LIN {X 0,Y 208.214,Z 248.661,A -85,B 0,C 180,E1 -22270.207,E2 -22270.207} C_VEL
LIN {X 0,Y 212.048,Z 236.781,A -85,B 0,C 180,E1 -22272.157,E2 -22272.157} C_VEL
LIN {X 0,Y 215.168,Z 224.656,A -85,B 0,C 180,E1 -22273.649,E2 -22273.649} C_VEL
LIN {X 0,Y 217.166,Z 214.19,A -85,B 0,C 180,E1 -22274.651,E2 -22274.651} C_VEL
LIN {X 0,Y 219.17,Z 200.943,A -85,B 0,C 180,E1 -22275.517,E2 -22275.517} C_VEL
LIN {X 0,Y 220.253,Z 187.914,A -85,B 0,C 180,E1 -22276.059,E2 -22276.059} C_VEL
LIN {X 0,Y 222.25,Z 151.476,A -85,B 0,C 180,E1 -22277.164,E2 -22277.164} C_VEL
LIN {X 0,Y 218.066,Z 142.469,A -85,B 0,C 180,E1 -22278.632,E2 -22278.632} C_VEL
LIN {X 0,Y 210.502,Z 129.434,A -85,B 0,C 180,E1 -22281.386,E2 -22281.386} C_VEL
LIN {X 0,Y 203.081,Z 118.196,A -85,B 0,C 180,E1 -22284.371,E2 -22284.371} C_VEL
LIN {X 0,Y 199.112,Z 112.832,A -85,B 0,C 180,E1 -22286.11,E2 -22286.11} C_VEL
LIN {X 0,Y 196.735,Z 109.497,A -85,B 0,C 180,E1 -22287.228,E2 -22287.228} C_VEL
LIN {X 0,Y 194.076,Z 106.045,A -85,B 0,C 180,E1 -22288.534,E2 -22288.534} C_VEL
LIN {X 0,Y 193.174,Z 104.766,A -85,B 0,C 180,E1 -22289.002,E2 -22289.002} C_VEL
LIN {X 0,Y 190.755,Z 102.14,A -85,B 0,C 180,E1 -22290.255,E2 -22290.255} C_VEL
LIN {X 0,Y 189.444,Z 99.842,A -85,B 0,C 180,E1 -22291.026,E2 -22291.026} C_VEL
LIN {X 0,Y 186.814,Z 97.643,A -85,B 0,C 180,E1 -22292.482,E2 -22292.482} C_VEL
LIN {X 0,Y 185.717,Z 95.405,A -85,B 0,C 180,E1 -22293.22,E2 -22293.22} C_VEL
LIN {X 0,Y 185.515,Z 94.365,A -85,B 0,C 180,E1 -22293.416,E2 -22293.416} C_VEL
LIN {X 0,Y 185.575,Z 94.354,A -85,B 0,C 180,E1 -22297.745,E2 -22297.745} C_VEL
LIN {X 0,Y 185.687,Z 94.337,A -85,B 0,C 180,E1 -22302.374,E2 -22302.374} C_VEL
LIN {X 0,Y 185.724,Z 94.335,A -85,B 0,C 180,E1 -22306.876,E2 -22306.876} C_VEL
LIN {X 0,Y 185.977,Z 94.319,A -85,B 0,C 180,E1 -22311.305,E2 -22311.305} C_VEL
LIN {X 0,Y 186.182,Z 94.286,A -85,B 0,C 180,E1 -22317.836,E2 -22317.836} C_VEL
LIN {X 0,Y 186.383,Z 94.246,A -85,B 0,C 180,E1 -22320,E2 -22320} C_VEL
LIN {X 0,Y 185.889,Z 94.317,A -85,B 0,C 180,E1 -22324.336,E2 -22324.336} C_VEL
LIN {X 0,Y 185.979,Z 94.318,A -85,B 0,C 180,E1 -22328.694,E2 -22328.694} C_VEL
LIN {X 0,Y 185.724,Z 94.335,A -85,B 0,C 180,E1 -22333.123,E2 -22333.123} C_VEL
LIN {X 0,Y 185.687,Z 94.336,A -85,B 0,C 180,E1 -22337.625,E2 -22337.625} C_VEL
LIN {X 0,Y 185.598,Z 94.35,A -85,B 0,C 180,E1 -22342.251,E2 -22342.251} C_VEL
LIN {X 0,Y 185.565,Z 94.357,A -85,B 0,C 180,E1 -22347.031,E2 -22347.031} C_VEL
LIN {X 0,Y 185.584,Z 94.473,A -85,B 0,C 180,E1 -22350.274,E2 -22350.274} C_VEL
LIN {X 0,Y 186.862,Z 98.544,A -85,B 0,C 180,E1 -22354.033,E2 -22354.033} C_VEL
LIN {X 0,Y 189.971,Z 103.26,A -85,B 0,C 180,E1 -22355.883,E2 -22355.883} C_VEL
LIN {X 0,Y 191.772,Z 105.585,A -85,B 0,C 180,E1 -22356.86,E2 -22356.86} C_VEL
LIN {X 0,Y 195.084,Z 110.421,A -85,B 0,C 180,E1 -22358.586,E2 -22358.586} C_VEL
LIN {X 0,Y 200.019,Z 118.409,A -85,B 0,C 180,E1 -22360.974,E2 -22360.974} C_VEL
LIN {X 0,Y 203.707,Z 124.608,A -85,B 0,C 180,E1 -22362.617,E2 -22362.617} C_VEL
LIN {X 0,Y 209.57,Z 135.23,A -85,B 0,C 180,E1 -22365.047,E2 -22365.047} C_VEL
LIN {X 0,Y 215.403,Z 147.492,A -85,B 0,C 180,E1 -22367.312,E2 -22367.312} C_VEL
LIN {X 0,Y 220.114,Z 159.014,A -85,B 0,C 180,E1 -22369.064,E2 -22369.064} C_VEL
LIN {X 0,Y 221.3,Z 169.331,A -85,B 0,C 180,E1 -22369.809,E2 -22369.809} C_VEL
LIN {X 0,Y 220.488,Z 184.555,A -85,B 0,C 180,E1 -22370.276,E2 -22370.276} C_VEL
LIN {X 0,Y 219.649,Z 190.415,A -85,B 0,C 180,E1 -22370.315,E2 -22370.315} C_VEL
LIN {X 0,Y 214.146,Z 209.415,A -85,B 0,C 180,E1 -22369.874,E2 -22369.874} C_VEL
LIN {X 0,Y 213.002,Z 215.173,A -85,B 0,C 180,E1 -22370.032,E2 -22370.032} C_VEL
LIN {X 0,Y 210.897,Z 228.271,A -85,B 0,C 180,E1 -22370.869,E2 -22370.869} C_VEL
LIN {X 0,Y 208.139,Z 240.343,A -85,B 0,C 180,E1 -22371.958,E2 -22371.958} C_VEL
LIN {X 0,Y 204.723,Z 251.98,A -85,B 0,C 180,E1 -22373.382,E2 -22373.382} C_VEL
LIN {X 0,Y 201.939,Z 260.097,A -85,B 0,C 180,E1 -22374.648,E2 -22374.648} C_VEL
LIN {X 0,Y 198.09,Z 270.178,A -85,B 0,C 180,E1 -22376.638,E2 -22376.638} C_VEL
LIN {X 0,Y 194.028,Z 279.294,A -85,B 0,C 180,E1 -22378.924,E2 -22378.924} C_VEL
LIN {X 0,Y 189.721,Z 288.196,A -85,B 0,C 180,E1 -22381.815,E2 -22381.815} C_VEL
LIN {X 0,Y 186.057,Z 295.38,A -85,B 0,C 180,E1 -22384.852,E2 -22384.852} C_VEL
LIN {X 0,Y 182.517,Z 301.95,A -85,B 0,C 180,E1 -22388.542,E2 -22388.542} C_VEL
LIN {X 0,Y 180.008,Z 306.321,A -85,B 0,C 180,E1 -22391.799,E2 -22391.799} C_VEL
LIN {X 0,Y 178.619,Z 308.644,A -85,B 0,C 180,E1 -22394.012,E2 -22394.012} C_VEL
LIN {X 0,Y 177.62,Z 310.548,A -85,B 0,C 180,E1 -22396.266,E2 -22396.266} C_VEL
LIN {X 0,Y 176.909,Z 311.998,A -85,B 0,C 180,E1 -22398.542,E2 -22398.542} C_VEL
LIN {X 0,Y 176.122,Z 313.708,A -85,B 0,C 180,E1 -22403.124,E2 -22403.124} C_VEL
LIN {X 0,Y 176.059,Z 313.961,A -85,B 0,C 180,E1 -22406.336,E2 -22406.336} C_VEL
LIN {X 0,Y 176.324,Z 313.298,A -85,B 0,C 180,E1 -22409.999,E2 -22409.999} C_VEL
LIN {X 0,Y 176.146,Z 311.28,A -85,B 0,C 180,E1 -22414.08,E2 -22414.08} C_VEL
LIN {X 0,Y 176.25,Z 308.042,A -85,B 0,C 180,E1 -22418.022,E2 -22418.022} C_VEL
LIN {X 0,Y 176.795,Z 304.072,A -85,B 0,C 180,E1 -22421.464,E2 -22421.464} C_VEL
LIN {X 0,Y 178.094,Z 297.957,A -85,B 0,C 180,E1 -22425.448,E2 -22425.448} C_VEL
LIN {X 0,Y 179.851,Z 291.253,A -85,B 0,C 180,E1 -22428.806,E2 -22428.806} C_VEL
LIN {X 0,Y 181.508,Z 285.685,A -85,B 0,C 180,E1 -22431.088,E2 -22431.088} C_VEL
LIN {X 0,Y 183.867,Z 276.18,A -85,B 0,C 180,E1 -22434.261,E2 -22434.261} C_VEL
LIN {X 0,Y 186.685,Z 266.151,A -85,B 0,C 180,E1 -22436.856,E2 -22436.856} C_VEL
LIN {X 0,Y 189.57,Z 254.816,A -85,B 0,C 180,E1 -22439.116,E2 -22439.116} C_VEL
LIN {X 0,Y 191.94,Z 243.68,A -85,B 0,C 180,E1 -22440.838,E2 -22440.838} C_VEL
LIN {X 0,Y 194.237,Z 231.337,A -85,B 0,C 180,E1 -22442.255,E2 -22442.255} C_VEL
LIN {X 0,Y 195.884,Z 218.597,A -85,B 0,C 180,E1 -22443.292,E2 -22443.292} C_VEL
LIN {X 0,Y 196.941,Z 205.474,A -85,B 0,C 180,E1 -22443.971,E2 -22443.971} C_VEL
LIN {X 0,Y 198.808,Z 161.492,A -85,B 0,C 180,E1 -22445.49,E2 -22445.49} C_VEL
LIN {X 0,Y 196.398,Z 137.184,A -85,B 0,C 180,E1 -22446.97,E2 -22446.97} C_VEL
LIN {X 0,Y 189.853,Z 120.576,A -85,B 0,C 180,E1 -22449.039,E2 -22449.039} C_VEL
LIN {X 0,Y 184.006,Z 108.494,A -85,B 0,C 180,E1 -22450.928,E2 -22450.928} C_VEL
LIN {X 0,Y 181.537,Z 103.873,A -85,B 0,C 180,E1 -22451.754,E2 -22451.754} C_VEL
LIN {X 0,Y 179.702,Z 100.17,A -85,B 0,C 180,E1 -22452.423,E2 -22452.423} C_VEL
LIN {X 0,Y 178.389,Z 95.265,A -85,B 0,C 180,E1 -22455.595,E2 -22455.595} C_VEL
LIN {X 0,Y 178.401,Z 95.258,A -85,B 0,C 180,E1 -22458.459,E2 -22458.459} C_VEL
LIN {X 0,Y 178.421,Z 95.248,A -85,B 0,C 180,E1 -22463.783,E2 -22463.783} C_VEL
LIN {X 0,Y 178.486,Z 95.25,A -85,B 0,C 180,E1 -22466.547,E2 -22466.547} C_VEL
LIN {X 0,Y 178.522,Z 95.247,A -85,B 0,C 180,E1 -22470.006,E2 -22470.006} C_VEL
LIN {X 0,Y 178.533,Z 95.24,A -85,B 0,C 180,E1 -22474.876,E2 -22474.876} C_VEL
LIN {X 0,Y 178.622,Z 95.22,A -85,B 0,C 180,E1 -22480.784,E2 -22480.784} C_VEL
LIN {X 0,Y 178.659,Z 95.214,A -85,B 0,C 180,E1 -22486.348,E2 -22486.348} C_VEL
LIN {X 0,Y 178.911,Z 95.199,A -85,B 0,C 180,E1 -22490.96,E2 -22490.96} C_VEL
LIN {X 0,Y 179.15,Z 95.157,A -85,B 0,C 180,E1 -22497.752,E2 -22497.752} C_VEL
LIN {X 0,Y 179.367,Z 95.142,A -85,B 0,C 180,E1 -22500,E2 -22500} C_VEL
LIN {X 0,Y 178.857,Z 95.184,A -85,B 0,C 180,E1 -22504.508,E2 -22504.508} C_VEL
LIN {X 0,Y 178.908,Z 95.196,A -85,B 0,C 180,E1 -22509.041,E2 -22509.041} C_VEL
LIN {X 0,Y 178.655,Z 95.209,A -85,B 0,C 180,E1 -22513.653,E2 -22513.653} C_VEL
LIN {X 0,Y 178.623,Z 95.225,A -85,B 0,C 180,E1 -22519.217,E2 -22519.217} C_VEL
LIN {X 0,Y 178.534,Z 95.245,A -85,B 0,C 180,E1 -22525.125,E2 -22525.125} C_VEL
LIN {X 0,Y 178.477,Z 95.25,A -85,B 0,C 180,E1 -22530.792,E2 -22530.792} C_VEL
LIN {X 0,Y 178.484,Z 95.251,A -85,B 0,C 180,E1 -22534.22,E2 -22534.22} C_VEL
LIN {X 0,Y 178.388,Z 95.265,A -85,B 0,C 180,E1 -22539.077,E2 -22539.077} C_VEL
LIN {X 0,Y 178.394,Z 95.262,A -85,B 0,C 180,E1 -22542.047,E2 -22542.047} C_VEL
LIN {X 0,Y 178.393,Z 95.263,A -85,B 0,C 180,E1 -22545.165,E2 -22545.165} C_VEL
LIN {X 0,Y 178.4,Z 95.263,A -85,B 0,C 180,E1 -22548.462,E2 -22548.462} C_VEL
LIN {X 0,Y 178.42,Z 95.261,A -85,B 0,C 180,E1 -22553.783,E2 -22553.783} C_VEL
LIN {X 0,Y 178.464,Z 95.409,A -85,B 0,C 180,E1 -22554.734,E2 -22554.734} C_VEL
LIN {X 0,Y 179.354,Z 97.939,A -85,B 0,C 180,E1 -22555.095,E2 -22555.095} C_VEL
LIN {X 0,Y 181.323,Z 100.58,A -85,B 0,C 180,E1 -22555.729,E2 -22555.729} C_VEL
LIN {X 0,Y 188.55,Z 112.687,A -85,B 0,C 180,E1 -22558.014,E2 -22558.014} C_VEL
LIN {X 0,Y 194.723,Z 124.313,A -85,B 0,C 180,E1 -22559.841,E2 -22559.841} C_VEL
LIN {X 0,Y 200.072,Z 136.131,A -85,B 0,C 180,E1 -22561.378,E2 -22561.378} C_VEL
LIN {X 0,Y 197.219,Z 194.928,A -85,B 0,C 180,E1 -22563.391,E2 -22563.391} C_VEL
LIN {X 0,Y 196.004,Z 208.238,A -85,B 0,C 180,E1 -22564.245,E2 -22564.245} C_VEL
LIN {X 0,Y 194.445,Z 220.579,A -85,B 0,C 180,E1 -22565.44,E2 -22565.44} C_VEL
LIN {X 0,Y 192.613,Z 231.72,A -85,B 0,C 180,E1 -22566.907,E2 -22566.907} C_VEL
LIN {X 0,Y 190.187,Z 243.267,A -85,B 0,C 180,E1 -22568.883,E2 -22568.883} C_VEL
LIN {X 0,Y 187.654,Z 253.66,A -85,B 0,C 180,E1 -22571.155,E2 -22571.155} C_VEL
LIN {X 0,Y 185.261,Z 262.174,A -85,B 0,C 180,E1 -22573.471,E2 -22573.471} C_VEL
LIN {X 0,Y 183.031,Z 270.012,A -85,B 0,C 180,E1 -22576.115,E2 -22576.115} C_VEL
LIN {X 0,Y 180.759,Z 277.681,A -85,B 0,C 180,E1 -22579.358,E2 -22579.358} C_VEL
LIN {X 0,Y 178.796,Z 284.725,A -85,B 0,C 180,E1 -22583.228,E2 -22583.228} C_VEL
LIN {X 0,Y 177.53,Z 289.43,A -85,B 0,C 180,E1 -22586.596,E2 -22586.596} C_VEL
LIN {X 0,Y 176.737,Z 293.036,A -85,B 0,C 180,E1 -22590.001,E2 -22590.001} C_VEL
LIN {X 0,Y 176.474,Z 294.901,A -85,B 0,C 180,E1 -22592.283,E2 -22592.283} C_VEL
LIN {X 0,Y 176.362,Z 296.496,A -85,B 0,C 180,E1 -22594.957,E2 -22594.957} C_VEL
LIN {X 0,Y 176.247,Z 297.954,A -85,B 0,C 180,E1 -22599.179,E2 -22599.179} C_VEL
LIN {X 0,Y 176.415,Z 298.2,A -85,B 0,C 180,E1 -22601.49,E2 -22601.49} C_VEL
LIN {X 0,Y 177.52,Z 297.423,A -85,B 0,C 180,E1 -22606.09,E2 -22606.09} C_VEL
LIN {X 0,Y 178.83,Z 295.862,A -85,B 0,C 180,E1 -22609.402,E2 -22609.402} C_VEL
LIN {X 0,Y 181.422,Z 292.147,A -85,B 0,C 180,E1 -22614.002,E2 -22614.002} C_VEL
LIN {X 0,Y 183.963,Z 288.165,A -85,B 0,C 180,E1 -22617.287,E2 -22617.287} C_VEL
LIN {X 0,Y 187.506,Z 282.086,A -85,B 0,C 180,E1 -22620.96,E2 -22620.96} C_VEL
LIN {X 0,Y 191.247,Z 275.216,A -85,B 0,C 180,E1 -22624.085,E2 -22624.085} C_VEL
LIN {X 0,Y 195.437,Z 266.754,A -85,B 0,C 180,E1 -22627.038,E2 -22627.038} C_VEL
LIN {X 0,Y 199.065,Z 257.983,A -85,B 0,C 180,E1 -22629.457,E2 -22629.457} C_VEL
LIN {X 0,Y 203.193,Z 247.149,A -85,B 0,C 180,E1 -22631.746,E2 -22631.746} C_VEL
LIN {X 0,Y 206.781,Z 236.268,A -85,B 0,C 180,E1 -22633.493,E2 -22633.493} C_VEL
LIN {X 0,Y 209.932,Z 224.261,A -85,B 0,C 180,E1 -22634.963,E2 -22634.963} C_VEL
LIN {X 0,Y 211.803,Z 214.817,A -85,B 0,C 180,E1 -22635.876,E2 -22635.876} C_VEL
LIN {X 0,Y 213.894,Z 201.6,A -85,B 0,C 180,E1 -22636.756,E2 -22636.756} C_VEL
LIN {X 0,Y 215.06,Z 188.275,A -85,B 0,C 180,E1 -22637.324,E2 -22637.324} C_VEL
LIN {X 0,Y 217.077,Z 153.919,A -85,B 0,C 180,E1 -22638.368,E2 -22638.368} C_VEL
LIN {X 0,Y 213.436,Z 146.148,A -85,B 0,C 180,E1 -22639.719,E2 -22639.719} C_VEL
LIN {X 0,Y 206.422,Z 134.012,A -85,B 0,C 180,E1 -22642.416,E2 -22642.416} C_VEL
LIN {X 0,Y 199.687,Z 123.62,A -85,B 0,C 180,E1 -22645.274,E2 -22645.274} C_VEL
LIN {X 0,Y 195.646,Z 117.975,A -85,B 0,C 180,E1 -22647.147,E2 -22647.147} C_VEL
LIN {X 0,Y 193.419,Z 114.948,A -85,B 0,C 180,E1 -22648.247,E2 -22648.247} C_VEL
LIN {X 0,Y 190.362,Z 110.778,A -85,B 0,C 180,E1 -22649.853,E2 -22649.853} C_VEL
LIN {X 0,Y 187.716,Z 107.553,A -85,B 0,C 180,E1 -22651.318,E2 -22651.318} C_VEL
LIN {X 0,Y 186.732,Z 106.033,A -85,B 0,C 180,E1 -22651.912,E2 -22651.912} C_VEL
LIN {X 0,Y 184.168,Z 103.462,A -85,B 0,C 180,E1 -22653.435,E2 -22653.435} C_VEL
LIN {X 0,Y 182.822,Z 100.932,A -85,B 0,C 180,E1 -22654.375,E2 -22654.375} C_VEL
LIN {X 0,Y 180.167,Z 98.955,A -85,B 0,C 180,E1 -22656.103,E2 -22656.103} C_VEL
LIN {X 0,Y 178.891,Z 96.811,A -85,B 0,C 180,E1 -22657.096,E2 -22657.096} C_VEL
LIN {X 0,Y 178.539,Z 95.229,A -85,B 0,C 180,E1 -22657.583,E2 -22657.583} C_VEL
LIN {X 0,Y 178.641,Z 95.216,A -85,B 0,C 180,E1 -22661.655,E2 -22661.655} C_VEL
LIN {X 0,Y 178.652,Z 95.22,A -85,B 0,C 180,E1 -22666.347,E2 -22666.347} C_VEL
LIN {X 0,Y 178.908,Z 95.2,A -85,B 0,C 180,E1 -22670.959,E2 -22670.959} C_VEL
LIN {X 0,Y 179.13,Z 95.165,A -85,B 0,C 180,E1 -22677.751,E2 -22677.751} C_VEL
LIN {X 0,Y 179.348,Z 95.122,A -85,B 0,C 180,E1 -22680,E2 -22680} C_VEL
LIN {X 0,Y 178.838,Z 95.193,A -85,B 0,C 180,E1 -22684.507,E2 -22684.507} C_VEL
LIN {X 0,Y 178.909,Z 95.199,A -85,B 0,C 180,E1 -22689.04,E2 -22689.04} C_VEL
LIN {X 0,Y 178.652,Z 95.221,A -85,B 0,C 180,E1 -22693.652,E2 -22693.652} C_VEL
LIN {X 0,Y 178.625,Z 95.229,A -85,B 0,C 180,E1 -22699.215,E2 -22699.215} C_VEL
LIN {X 0,Y 178.537,Z 95.243,A -85,B 0,C 180,E1 -22705.124,E2 -22705.124} C_VEL
LIN {X 0,Y 178.515,Z 95.236,A -85,B 0,C 180,E1 -22706.92,E2 -22706.92} C_VEL
LIN {X 0,Y 179.396,Z 97.872,A -85,B 0,C 180,E1 -22709.746,E2 -22709.746} C_VEL
LIN {X 0,Y 182.55,Z 102.601,A -85,B 0,C 180,E1 -22712.028,E2 -22712.028} C_VEL
LIN {X 0,Y 184.519,Z 105.013,A -85,B 0,C 180,E1 -22713.295,E2 -22713.295} C_VEL
LIN {X 0,Y 188.306,Z 110.4,A -85,B 0,C 180,E1 -22715.59,E2 -22715.59} C_VEL
LIN {X 0,Y 192.963,Z 117.683,A -85,B 0,C 180,E1 -22718.16,E2 -22718.16} C_VEL
LIN {X 0,Y 197.039,Z 124.388,A -85,B 0,C 180,E1 -22720.206,E2 -22720.206} C_VEL
LIN {X 0,Y 201.68,Z 132.442,A -85,B 0,C 180,E1 -22722.352,E2 -22722.352} C_VEL
LIN {X 0,Y 207.554,Z 143.812,A -85,B 0,C 180,E1 -22724.866,E2 -22724.866} C_VEL
LIN {X 0,Y 213.318,Z 157.114,A -85,B 0,C 180,E1 -22727.195,E2 -22727.195} C_VEL
LIN {X 0,Y 215.175,Z 161.886,A -85,B 0,C 180,E1 -22727.921,E2 -22727.921} C_VEL
LIN {X 0,Y 216.084,Z 170.94,A -85,B 0,C 180,E1 -22728.576,E2 -22728.576} C_VEL
LIN {X 0,Y 213.683,Z 209.608,A -85,B 0,C 180,E1 -22729.791,E2 -22729.791} C_VEL
LIN {X 0,Y 213.002,Z 215.173,A -85,B 0,C 180,E1 -22730.032,E2 -22730.032} C_VEL
LIN {X 0,Y 212.19,Z 218.992,A -85,B 0,C 180,E1 -22730.167,E2 -22730.167} C_VEL
LIN {X 0,Y 209.468,Z 226.416,A -85,B 0,C 180,E1 -22730.29,E2 -22730.29} C_VEL
LIN {X 0,Y 203.966,Z 238.08,A -85,B 0,C 180,E1 -22730.587,E2 -22730.587} C_VEL
LIN {X 0,Y 201.638,Z 244.264,A -85,B 0,C 180,E1 -22731.113,E2 -22731.113} C_VEL
LIN {X 0,Y 198.06,Z 255.152,A -85,B 0,C 180,E1 -22732.578,E2 -22732.578} C_VEL
LIN {X 0,Y 193.935,Z 266.11,A -85,B 0,C 180,E1 -22734.561,E2 -22734.561} C_VEL
LIN {X 0,Y 189.672,Z 275.927,A -85,B 0,C 180,E1 -22736.869,E2 -22736.869} C_VEL
LIN {X 0,Y 185.67,Z 283.993,A -85,B 0,C 180,E1 -22739.269,E2 -22739.269} C_VEL
LIN {X 0,Y 181.418,Z 291.932,A -85,B 0,C 180,E1 -22742.297,E2 -22742.297} C_VEL
LIN {X 0,Y 178.037,Z 298.141,A -85,B 0,C 180,E1 -22745.403,E2 -22745.403} C_VEL
LIN {X 0,Y 174.926,Z 303.391,A -85,B 0,C 180,E1 -22748.801,E2 -22748.801} C_VEL
LIN {X 0,Y 172.511,Z 307.361,A -85,B 0,C 180,E1 -22752.208,E2 -22752.208} C_VEL
LIN {X 0,Y 170.684,Z 310.316,A -85,B 0,C 180,E1 -22755.696,E2 -22755.696} C_VEL
LIN {X 0,Y 169.355,Z 312.766,A -85,B 0,C 180,E1 -22760.444,E2 -22760.444} C_VEL
LIN {X 0,Y 168.966,Z 313.672,A -85,B 0,C 180,E1 -22765.227,E2 -22765.227} C_VEL
LIN {X 0,Y 169.054,Z 313.501,A -85,B 0,C 180,E1 -22767.617,E2 -22767.617} C_VEL
LIN {X 0,Y 169.24,Z 312.933,A -85,B 0,C 180,E1 -22769.999,E2 -22769.999} C_VEL
LIN {X 0,Y 169.056,Z 311.115,A -85,B 0,C 180,E1 -22773.863,E2 -22773.863} C_VEL
LIN {X 0,Y 169.185,Z 307.6,A -85,B 0,C 180,E1 -22778.359,E2 -22778.359} C_VEL
LIN {X 0,Y 169.78,Z 303.588,A -85,B 0,C 180,E1 -22781.944,E2 -22781.944} C_VEL
LIN {X 0,Y 171.235,Z 297.41,A -85,B 0,C 180,E1 -22786.083,E2 -22786.083} C_VEL
LIN {X 0,Y 173.109,Z 290.654,A -85,B 0,C 180,E1 -22789.568,E2 -22789.568} C_VEL
LIN {X 0,Y 174.701,Z 285.446,A -85,B 0,C 180,E1 -22791.777,E2 -22791.777} C_VEL
LIN {X 0,Y 176.871,Z 277.26,A -85,B 0,C 180,E1 -22794.658,E2 -22794.658} C_VEL
LIN {X 0,Y 179.713,Z 267.506,A -85,B 0,C 180,E1 -22797.355,E2 -22797.355} C_VEL
LIN {X 0,Y 182.663,Z 256.674,A -85,B 0,C 180,E1 -22799.693,E2 -22799.693} C_VEL
LIN {X 0,Y 185.094,Z 246.118,A -85,B 0,C 180,E1 -22801.472,E2 -22801.472} C_VEL
LIN {X 0,Y 187.645,Z 233.414,A -85,B 0,C 180,E1 -22803.053,E2 -22803.053} C_VEL
LIN {X 0,Y 189.537,Z 220.471,A -85,B 0,C 180,E1 -22804.216,E2 -22804.216} C_VEL
LIN {X 0,Y 190.723,Z 207.67,A -85,B 0,C 180,E1 -22804.961,E2 -22804.961} C_VEL
LIN {X 0,Y 192.809,Z 162.477,A -85,B 0,C 180,E1 -22806.567,E2 -22806.567} C_VEL
LIN {X 0,Y 190.647,Z 139.752,A -85,B 0,C 180,E1 -22808.004,E2 -22808.004} C_VEL
LIN {X 0,Y 185.116,Z 125.198,A -85,B 0,C 180,E1 -22809.873,E2 -22809.873} C_VEL
LIN {X 0,Y 179.303,Z 112.892,A -85,B 0,C 180,E1 -22811.865,E2 -22811.865} C_VEL
LIN {X 0,Y 174.268,Z 103.614,A -85,B 0,C 180,E1 -22813.673,E2 -22813.673} C_VEL
LIN {X 0,Y 172.282,Z 99.694,A -85,B 0,C 180,E1 -22814.494,E2 -22814.494} C_VEL
LIN {X 0,Y 171.354,Z 96.14,A -85,B 0,C 180,E1 -22816.917,E2 -22816.917} C_VEL
LIN {X 0,Y 171.363,Z 96.108,A -85,B 0,C 180,E1 -22822.035,E2 -22822.035} C_VEL
LIN {X 0,Y 171.397,Z 96.134,A -85,B 0,C 180,E1 -22825.092,E2 -22825.092} C_VEL
LIN {X 0,Y 171.448,Z 96.129,A -85,B 0,C 180,E1 -22830.535,E2 -22830.535} C_VEL
LIN {X 0,Y 171.457,Z 96.127,A -85,B 0,C 180,E1 -22835.802,E2 -22835.802} C_VEL
LIN {X 0,Y 171.578,Z 96.097,A -85,B 0,C 180,E1 -22840.872,E2 -22840.872} C_VEL
LIN {X 0,Y 171.577,Z 96.101,A -85,B 0,C 180,E1 -22845.773,E2 -22845.773} C_VEL
LIN {X 0,Y 171.847,Z 96.075,A -85,B 0,C 180,E1 -22850.585,E2 -22850.585} C_VEL
LIN {X 0,Y 171.811,Z 96.066,A -85,B 0,C 180,E1 -22855.308,E2 -22855.308} C_VEL
LIN {X 0,Y 172.33,Z 96.018,A -85,B 0,C 180,E1 -22860.001,E2 -22860.001} C_VEL
LIN {X 0,Y 171.805,Z 96.061,A -85,B 0,C 180,E1 -22864.693,E2 -22864.693} C_VEL
LIN {X 0,Y 171.845,Z 96.077,A -85,B 0,C 180,E1 -22869.416,E2 -22869.416} C_VEL
LIN {X 0,Y 171.573,Z 96.093,A -85,B 0,C 180,E1 -22874.228,E2 -22874.228} C_VEL
LIN {X 0,Y 171.545,Z 96.104,A -85,B 0,C 180,E1 -22879.563,E2 -22879.563} C_VEL
LIN {X 0,Y 171.469,Z 96.125,A -85,B 0,C 180,E1 -22885.617,E2 -22885.617} C_VEL
LIN {X 0,Y 171.44,Z 96.127,A -85,B 0,C 180,E1 -22890.587,E2 -22890.587} C_VEL
LIN {X 0,Y 171.392,Z 96.133,A -85,B 0,C 180,E1 -22895.036,E2 -22895.036} C_VEL
LIN {X 0,Y 171.344,Z 96.14,A -85,B 0,C 180,E1 -22898.803,E2 -22898.803} C_VEL
LIN {X 0,Y 171.319,Z 96.144,A -85,B 0,C 180,E1 -22904.219,E2 -22904.219} C_VEL
LIN {X 0,Y 171.332,Z 96.144,A -85,B 0,C 180,E1 -22908.981,E2 -22908.981} C_VEL
LIN {X 0,Y 171.348,Z 96.148,A -85,B 0,C 180,E1 -22912.791,E2 -22912.791} C_VEL
LIN {X 0,Y 172.434,Z 99.112,A -85,B 0,C 180,E1 -22913.268,E2 -22913.268} C_VEL
LIN {X 0,Y 174.241,Z 101.349,A -85,B 0,C 180,E1 -22913.898,E2 -22913.898} C_VEL
LIN {X 0,Y 176.435,Z 104.7,A -85,B 0,C 180,E1 -22914.673,E2 -22914.673} C_VEL
LIN {X 0,Y 183.024,Z 115.736,A -85,B 0,C 180,E1 -22916.888,E2 -22916.888} C_VEL
LIN {X 0,Y 189.243,Z 127.483,A -85,B 0,C 180,E1 -22918.845,E2 -22918.845} C_VEL
LIN {X 0,Y 194.018,Z 137.872,A -85,B 0,C 180,E1 -22920.294,E2 -22920.294} C_VEL
LIN {X 0,Y 191.167,Z 194.962,A -85,B 0,C 180,E1 -22922.297,E2 -22922.297} C_VEL
LIN {X 0,Y 189.934,Z 208.269,A -85,B 0,C 180,E1 -22923.169,E2 -22923.169} C_VEL
LIN {X 0,Y 188.241,Z 221,A -85,B 0,C 180,E1 -22924.426,E2 -22924.426} C_VEL
LIN {X 0,Y 186.15,Z 232.898,A -85,B 0,C 180,E1 -22926.056,E2 -22926.056} C_VEL
LIN {X 0,Y 183.624,Z 244.288,A -85,B 0,C 180,E1 -22928.089,E2 -22928.089} C_VEL
LIN {X 0,Y 180.983,Z 254.561,A -85,B 0,C 180,E1 -22930.432,E2 -22930.432} C_VEL
LIN {X 0,Y 178.5,Z 262.976,A -85,B 0,C 180,E1 -22932.826,E2 -22932.826} C_VEL
LIN {X 0,Y 175.779,Z 272.078,A -85,B 0,C 180,E1 -22936.121,E2 -22936.121} C_VEL
LIN {X 0,Y 173.468,Z 279.413,A -85,B 0,C 180,E1 -22939.496,E2 -22939.496} C_VEL
LIN {X 0,Y 171.775,Z 285.291,A -85,B 0,C 180,E1 -22942.95,E2 -22942.95} C_VEL
LIN {X 0,Y 170.445,Z 289.945,A -85,B 0,C 180,E1 -22946.455,E2 -22946.455} C_VEL
LIN {X 0,Y 169.656,Z 293.501,A -85,B 0,C 180,E1 -22950.001,E2 -22950.001} C_VEL
LIN {X 0,Y 169.384,Z 295.33,A -85,B 0,C 180,E1 -22952.379,E2 -22952.379} C_VEL
LIN {X 0,Y 169.289,Z 296.76,A -85,B 0,C 180,E1 -22954.884,E2 -22954.884} C_VEL
LIN {X 0,Y 169.188,Z 298.31,A -85,B 0,C 180,E1 -22959.565,E2 -22959.565} C_VEL
LIN {X 0,Y 169.401,Z 298.519,A -85,B 0,C 180,E1 -22961.973,E2 -22961.973} C_VEL
LIN {X 0,Y 170.627,Z 297.691,A -85,B 0,C 180,E1 -22966.758,E2 -22966.758} C_VEL
LIN {X 0,Y 171.922,Z 296.261,A -85,B 0,C 180,E1 -22969.909,E2 -22969.909} C_VEL
LIN {X 0,Y 174.071,Z 293.388,A -85,B 0,C 180,E1 -22973.813,E2 -22973.813} C_VEL
LIN {X 0,Y 176.597,Z 289.721,A -85,B 0,C 180,E1 -22977.237,E2 -22977.237} C_VEL
LIN {X 0,Y 179.678,Z 284.827,A -85,B 0,C 180,E1 -22980.624,E2 -22980.624} C_VEL
LIN {X 0,Y 183.312,Z 278.804,A -85,B 0,C 180,E1 -22983.775,E2 -22983.775} C_VEL
LIN {X 0,Y 187.459,Z 271.177,A -85,B 0,C 180,E1 -22986.86,E2 -22986.86} C_VEL
LIN {X 0,Y 191.611,Z 262.34,A -85,B 0,C 180,E1 -22989.623,E2 -22989.623} C_VEL
LIN {X 0,Y 195.688,Z 252.605,A -85,B 0,C 180,E1 -22991.984,E2 -22991.984} C_VEL
LIN {X 0,Y 199.765,Z 241.619,A -85,B 0,C 180,E1 -22994.015,E2 -22994.015} C_VEL
LIN {X 0,Y 203.067,Z 230.797,A -85,B 0,C 180,E1 -22995.547,E2 -22995.547} C_VEL
LIN {X 0,Y 205.919,Z 218.39,A -85,B 0,C 180,E1 -22996.915,E2 -22996.915} C_VEL
LIN {X 0,Y 208.258,Z 205.643,A -85,B 0,C 180,E1 -22997.871,E2 -22997.871} C_VEL
LIN {X 0,Y 209.754,Z 191.86,A -85,B 0,C 180,E1 -22998.538,E2 -22998.538} C_VEL
LIN {X 0,Y 211.924,Z 156.256,A -85,B 0,C 180,E1 -22999.659,E2 -22999.659} C_VEL
LIN {X 0,Y 208.539,Z 149.298,A -85,B 0,C 180,E1 -23000.983,E2 -23000.983} C_VEL
LIN {X 0,Y 202.366,Z 138.531,A -85,B 0,C 180,E1 -23003.505,E2 -23003.505} C_VEL
LIN {X 0,Y 196.398,Z 129.041,A -85,B 0,C 180,E1 -23006.189,E2 -23006.189} C_VEL
LIN {X 0,Y 190.681,Z 120.93,A -85,B 0,C 180,E1 -23009.038,E2 -23009.038} C_VEL
LIN {X 0,Y 187.427,Z 116.547,A -85,B 0,C 180,E1 -23010.825,E2 -23010.825} C_VEL
LIN {X 0,Y 184.56,Z 112.583,A -85,B 0,C 180,E1 -23012.539,E2 -23012.539} C_VEL
LIN {X 0,Y 181.574,Z 109.281,A -85,B 0,C 180,E1 -23014.417,E2 -23014.417} C_VEL
LIN {X 0,Y 180.462,Z 107.364,A -85,B 0,C 180,E1 -23015.218,E2 -23015.218} C_VEL
LIN {X 0,Y 177.688,Z 104.843,A -85,B 0,C 180,E1 -23017.162,E2 -23017.162} C_VEL
LIN {X 0,Y 176.125,Z 101.923,A -85,B 0,C 180,E1 -23018.492,E2 -23018.492} C_VEL
LIN {X 0,Y 173.471,Z 100.142,A -85,B 0,C 180,E1 -23020.646,E2 -23020.646} C_VEL
LIN {X 0,Y 171.913,Z 97.508,A -85,B 0,C 180,E1 -23022.221,E2 -23022.221} C_VEL
LIN {X 0,Y 171.573,Z 96.095,A -85,B 0,C 180,E1 -23022.723,E2 -23022.723} C_VEL
LIN {X 0,Y 171.771,Z 96.072,A -85,B 0,C 180,E1 -23029.105,E2 -23029.105} C_VEL
LIN {X 0,Y 171.862,Z 96.058,A -85,B 0,C 180,E1 -23032.953,E2 -23032.953} C_VEL
LIN {X 0,Y 172.078,Z 96.044,A -85,B 0,C 180,E1 -23037.659,E2 -23037.659} C_VEL
LIN {X 0,Y 172.313,Z 95.998,A -85,B 0,C 180,E1 -23039.999,E2 -23039.999} C_VEL
LIN {X 0,Y 171.788,Z 96.069,A -85,B 0,C 180,E1 -23044.693,E2 -23044.693} C_VEL
LIN {X 0,Y 171.847,Z 96.075,A -85,B 0,C 180,E1 -23049.415,E2 -23049.415} C_VEL
LIN {X 0,Y 171.57,Z 96.11,A -85,B 0,C 180,E1 -23054.227,E2 -23054.227} C_VEL
LIN {X 0,Y 171.547,Z 96.114,A -85,B 0,C 180,E1 -23059.561,E2 -23059.561} C_VEL
LIN {X 0,Y 171.476,Z 96.224,A -85,B 0,C 180,E1 -23063.074,E2 -23063.074} C_VEL
LIN {X 0,Y 171.649,Z 97.109,A -85,B 0,C 180,E1 -23063.928,E2 -23063.928} C_VEL
LIN {X 0,Y 172.809,Z 99.431,A -85,B 0,C 180,E1 -23065.17,E2 -23065.17} C_VEL
LIN {X 0,Y 175.227,Z 102.077,A -85,B 0,C 180,E1 -23067.305,E2 -23067.305} C_VEL
LIN {X 0,Y 177.459,Z 104.562,A -85,B 0,C 180,E1 -23069.086,E2 -23069.086} C_VEL
LIN {X 0,Y 180.784,Z 109.421,A -85,B 0,C 180,E1 -23071.564,E2 -23071.564} C_VEL
LIN {X 0,Y 182.157,Z 111.288,A -85,B 0,C 180,E1 -23072.495,E2 -23072.495} C_VEL
LIN {X 0,Y 186.372,Z 117.641,A -85,B 0,C 180,E1 -23075.166,E2 -23075.166} C_VEL
LIN {X 0,Y 189.961,Z 123.35,A -85,B 0,C 180,E1 -23077.228,E2 -23077.228} C_VEL
LIN {X 0,Y 194.422,Z 130.891,A -85,B 0,C 180,E1 -23079.576,E2 -23079.576} C_VEL
LIN {X 0,Y 199.954,Z 141.009,A -85,B 0,C 180,E1 -23082.226,E2 -23082.226} C_VEL
LIN {X 0,Y 205.439,Z 152.708,A -85,B 0,C 180,E1 -23084.667,E2 -23084.667} C_VEL
LIN {X 0,Y 209.917,Z 163.668,A -85,B 0,C 180,E1 -23086.555,E2 -23086.555} C_VEL
LIN {X 0,Y 210.479,Z 166.241,A -85,B 0,C 180,E1 -23086.839,E2 -23086.839} C_VEL
LIN {X 0,Y 211.026,Z 171.734,A -85,B 0,C 180,E1 -23087.256,E2 -23087.256} C_VEL
LIN {X 0,Y 208.598,Z 209.096,A -85,B 0,C 180,E1 -23088.44,E2 -23088.44} C_VEL
LIN {X 0,Y 206.768,Z 222.364,A -85,B 0,C 180,E1 -23089.142,E2 -23089.142} C_VEL
LIN {X 0,Y 204.176,Z 234.897,A -85,B 0,C 180,E1 -23090.126,E2 -23090.126} C_VEL
LIN {X 0,Y 201.638,Z 244.264,A -85,B 0,C 180,E1 -23091.113,E2 -23091.113} C_VEL
LIN {X 0,Y 200.038,Z 247.795,A -85,B 0,C 180,E1 -23091.411,E2 -23091.411} C_VEL
LIN {X 0,Y 192.222,Z 257.923,A -85,B 0,C 180,E1 -23091.866,E2 -23091.866} C_VEL
LIN {X 0,Y 190.363,Z 261.133,A -85,B 0,C 180,E1 -23092.295,E2 -23092.295} C_VEL
LIN {X 0,Y 190.153,Z 261.657,A -85,B 0,C 180,E1 -23092.397,E2 -23092.397} C_VEL
LIN {X 0,Y 185.507,Z 272.367,A -85,B 0,C 180,E1 -23094.707,E2 -23094.707} C_VEL
LIN {X 0,Y 181.206,Z 281.012,A -85,B 0,C 180,E1 -23097.112,E2 -23097.112} C_VEL
LIN {X 0,Y 176.581,Z 289.423,A -85,B 0,C 180,E1 -23100.164,E2 -23100.164} C_VEL
LIN {X 0,Y 172.654,Z 296.214,A -85,B 0,C 180,E1 -23103.399,E2 -23103.399} C_VEL
LIN {X 0,Y 169.358,Z 301.668,A -85,B 0,C 180,E1 -23106.781,E2 -23106.781} C_VEL
LIN {X 0,Y 166.553,Z 305.955,A -85,B 0,C 180,E1 -23110.27,E2 -23110.27} C_VEL
LIN {X 0,Y 164.989,Z 308.238,A -85,B 0,C 180,E1 -23112.651,E2 -23112.651} C_VEL
LIN {X 0,Y 163.77,Z 310.077,A -85,B 0,C 180,E1 -23115.078,E2 -23115.078} C_VEL
LIN {X 0,Y 162.34,Z 312.489,A -85,B 0,C 180,E1 -23120.027,E2 -23120.027} C_VEL
LIN {X 0,Y 161.885,Z 313.348,A -85,B 0,C 180,E1 -23125.018,E2 -23125.018} C_VEL
LIN {X 0,Y 161.973,Z 313.154,A -85,B 0,C 180,E1 -23127.512,E2 -23127.512} C_VEL
LIN {X 0,Y 162.159,Z 312.568,A -85,B 0,C 180,E1 -23129.999,E2 -23129.999} C_VEL
LIN {X 0,Y 161.986,Z 310.892,A -85,B 0,C 180,E1 -23133.729,E2 -23133.729} C_VEL
LIN {X 0,Y 162.143,Z 307.154,A -85,B 0,C 180,E1 -23138.725,E2 -23138.725} C_VEL
LIN {X 0,Y 162.793,Z 303.1,A -85,B 0,C 180,E1 -23142.465,E2 -23142.465} C_VEL
LIN {X 0,Y 164.395,Z 296.862,A -85,B 0,C 180,E1 -23146.771,E2 -23146.771} C_VEL
LIN {X 0,Y 166.412,Z 290.057,A -85,B 0,C 180,E1 -23150.39,E2 -23150.39} C_VEL
LIN {X 0,Y 168.671,Z 282.56,A -85,B 0,C 180,E1 -23153.556,E2 -23153.556} C_VEL
LIN {X 0,Y 170.919,Z 274.732,A -85,B 0,C 180,E1 -23156.233,E2 -23156.233} C_VEL
LIN {X 0,Y 174.029,Z 264.485,A -85,B 0,C 180,E1 -23158.986,E2 -23158.986} C_VEL
LIN {X 0,Y 177.257,Z 252.894,A -85,B 0,C 180,E1 -23161.358,E2 -23161.358} C_VEL
LIN {X 0,Y 179.874,Z 241.454,A -85,B 0,C 180,E1 -23163.161,E2 -23163.161} C_VEL
LIN {X 0,Y 182.142,Z 229.71,A -85,B 0,C 180,E1 -23164.521,E2 -23164.521} C_VEL
LIN {X 0,Y 183.941,Z 216.08,A -85,B 0,C 180,E1 -23165.64,E2 -23165.64} C_VEL
LIN {X 0,Y 184.945,Z 203.329,A -85,B 0,C 180,E1 -23166.293,E2 -23166.293} C_VEL
LIN {X 0,Y 186.893,Z 163.668,A -85,B 0,C 180,E1 -23167.701,E2 -23167.701} C_VEL
LIN {X 0,Y 184.922,Z 141.814,A -85,B 0,C 180,E1 -23169.134,E2 -23169.134} C_VEL
LIN {X 0,Y 178.457,Z 125.307,A -85,B 0,C 180,E1 -23171.455,E2 -23171.455} C_VEL
LIN {X 0,Y 172.466,Z 113.061,A -85,B 0,C 180,E1 -23173.672,E2 -23173.672} C_VEL
LIN {X 0,Y 167.298,Z 103.786,A -85,B 0,C 180,E1 -23175.702,E2 -23175.702} C_VEL
LIN {X 0,Y 164.938,Z 99.196,A -85,B 0,C 180,E1 -23176.81,E2 -23176.81} C_VEL
LIN {X 0,Y 164.282,Z 97.012,A -85,B 0,C 180,E1 -23178.464,E2 -23178.464} C_VEL
LIN {X 0,Y 164.325,Z 97.008,A -85,B 0,C 180,E1 -23184.35,E2 -23184.35} C_VEL
LIN {X 0,Y 164.39,Z 97.006,A -85,B 0,C 180,E1 -23189.135,E2 -23189.135} C_VEL
LIN {X 0,Y 164.415,Z 96.997,A -85,B 0,C 180,E1 -23194.694,E2 -23194.694} C_VEL
LIN {X 0,Y 164.483,Z 96.977,A -85,B 0,C 180,E1 -23200.051,E2 -23200.051} C_VEL
LIN {X 0,Y 164.524,Z 96.985,A -85,B 0,C 180,E1 -23205.15,E2 -23205.15} C_VEL
LIN {X 0,Y 164.767,Z 96.954,A -85,B 0,C 180,E1 -23210.177,E2 -23210.177} C_VEL
LIN {X 0,Y 164.83,Z 96.952,A -85,B 0,C 180,E1 -23212.651,E2 -23212.651} C_VEL
LIN {X 0,Y 165.045,Z 96.911,A -85,B 0,C 180,E1 -23217.56,E2 -23217.56} C_VEL
LIN {X 0,Y 165.292,Z 96.894,A -85,B 0,C 180,E1 -23220.001,E2 -23220.001} C_VEL
LIN {X 0,Y 164.754,Z 96.938,A -85,B 0,C 180,E1 -23224.895,E2 -23224.895} C_VEL
LIN {X 0,Y 164.825,Z 96.946,A -85,B 0,C 180,E1 -23227.35,E2 -23227.35} C_VEL
LIN {X 0,Y 164.702,Z 96.956,A -85,B 0,C 180,E1 -23231.061,E2 -23231.061} C_VEL
LIN {X 0,Y 164.483,Z 96.994,A -85,B 0,C 180,E1 -23237.404,E2 -23237.404} C_VEL
LIN {X 0,Y 164.473,Z 96.981,A -85,B 0,C 180,E1 -23239.99,E2 -23239.99} C_VEL
LIN {X 0,Y 164.393,Z 97.005,A -85,B 0,C 180,E1 -23246.134,E2 -23246.134} C_VEL
LIN {X 0,Y 164.374,Z 97.006,A -85,B 0,C 180,E1 -23251.228,E2 -23251.228} C_VEL
LIN {X 0,Y 164.28,Z 97.023,A -85,B 0,C 180,E1 -23256.794,E2 -23256.794} C_VEL
LIN {X 0,Y 164.286,Z 97.022,A -85,B 0,C 180,E1 -23259.919,E2 -23259.919} C_VEL
LIN {X 0,Y 164.28,Z 97.023,A -85,B 0,C 180,E1 -23263.343,E2 -23263.343} C_VEL
LIN {X 0,Y 164.262,Z 97.023,A -85,B 0,C 180,E1 -23266.8,E2 -23266.8} C_VEL
LIN {X 0,Y 164.276,Z 97.052,A -85,B 0,C 180,E1 -23270.641,E2 -23270.641} C_VEL
LIN {X 0,Y 165.239,Z 99.743,A -85,B 0,C 180,E1 -23271.113,E2 -23271.113} C_VEL
LIN {X 0,Y 167.348,Z 102.373,A -85,B 0,C 180,E1 -23271.932,E2 -23271.932} C_VEL
LIN {X 0,Y 169.461,Z 105.646,A -85,B 0,C 180,E1 -23272.757,E2 -23272.757} C_VEL
LIN {X 0,Y 176.371,Z 116.677,A -85,B 0,C 180,E1 -23275.273,E2 -23275.273} C_VEL
LIN {X 0,Y 183.766,Z 130.486,A -85,B 0,C 180,E1 -23277.77,E2 -23277.77} C_VEL
LIN {X 0,Y 188.042,Z 139.869,A -85,B 0,C 180,E1 -23279.154,E2 -23279.154} C_VEL
LIN {X 0,Y 185.139,Z 195.727,A -85,B 0,C 180,E1 -23281.176,E2 -23281.176} C_VEL
LIN {X 0,Y 183.759,Z 209.387,A -85,B 0,C 180,E1 -23282.104,E2 -23282.104} C_VEL
LIN {X 0,Y 181.955,Z 222.425,A -85,B 0,C 180,E1 -23283.475,E2 -23283.475} C_VEL
LIN {X 0,Y 179.732,Z 234.069,A -85,B 0,C 180,E1 -23285.144,E2 -23285.144} C_VEL
LIN {X 0,Y 177.099,Z 245.304,A -85,B 0,C 180,E1 -23287.238,E2 -23287.238} C_VEL
LIN {X 0,Y 174.345,Z 255.442,A -85,B 0,C 180,E1 -23289.655,E2 -23289.655} C_VEL
LIN {X 0,Y 171.25,Z 265.377,A -85,B 0,C 180,E1 -23292.691,E2 -23292.691} C_VEL
LIN {X 0,Y 168.474,Z 274.113,A -85,B 0,C 180,E1 -23296.122,E2 -23296.122} C_VEL
LIN {X 0,Y 166.185,Z 281.11,A -85,B 0,C 180,E1 -23299.646,E2 -23299.646} C_VEL
LIN {X 0,Y 164.277,Z 287.495,A -85,B 0,C 180,E1 -23303.861,E2 -23303.861} C_VEL
LIN {X 0,Y 163.023,Z 291.725,A -85,B 0,C 180,E1 -23307.53,E2 -23307.53} C_VEL
LIN {X 0,Y 162.577,Z 293.965,A -85,B 0,C 180,E1 -23310.001,E2 -23310.001} C_VEL
LIN {X 0,Y 162.278,Z 295.751,A -85,B 0,C 180,E1 -23312.483,E2 -23312.483} C_VEL
LIN {X 0,Y 162.179,Z 297.102,A -85,B 0,C 180,E1 -23314.973,E2 -23314.973} C_VEL
LIN {X 0,Y 162.118,Z 298.667,A -85,B 0,C 180,E1 -23319.987,E2 -23319.987} C_VEL
LIN {X 0,Y 162.387,Z 298.832,A -85,B 0,C 180,E1 -23322.498,E2 -23322.498} C_VEL
LIN {X 0,Y 163.743,Z 297.961,A -85,B 0,C 180,E1 -23327.485,E2 -23327.485} C_VEL
LIN {X 0,Y 165.028,Z 296.662,A -85,B 0,C 180,E1 -23330.459,E2 -23330.459} C_VEL
LIN {X 0,Y 167.497,Z 293.567,A -85,B 0,C 180,E1 -23334.809,E2 -23334.809} C_VEL
LIN {X 0,Y 170.216,Z 289.851,A -85,B 0,C 180,E1 -23338.348,E2 -23338.348} C_VEL
LIN {X 0,Y 173.476,Z 284.988,A -85,B 0,C 180,E1 -23341.781,E2 -23341.781} C_VEL
LIN {X 0,Y 177.372,Z 278.825,A -85,B 0,C 180,E1 -23345.068,E2 -23345.068} C_VEL
LIN {X 0,Y 181.754,Z 271.107,A -85,B 0,C 180,E1 -23348.221,E2 -23348.221} C_VEL
LIN {X 0,Y 185.727,Z 262.996,A -85,B 0,C 180,E1 -23350.815,E2 -23350.815} C_VEL
LIN {X 0,Y 189.943,Z 253.423,A -85,B 0,C 180,E1 -23353.198,E2 -23353.198} C_VEL
LIN {X 0,Y 194.182,Z 242.57,A -85,B 0,C 180,E1 -23355.259,E2 -23355.259} C_VEL
LIN {X 0,Y 197.605,Z 231.941,A -85,B 0,C 180,E1 -23356.812,E2 -23356.812} C_VEL
LIN {X 0,Y 200.445,Z 220.338,A -85,B 0,C 180,E1 -23358.142,E2 -23358.142} C_VEL
LIN {X 0,Y 203.026,Z 206.999,A -85,B 0,C 180,E1 -23359.201,E2 -23359.201} C_VEL
LIN {X 0,Y 204.625,Z 194.401,A -85,B 0,C 180,E1 -23359.846,E2 -23359.846} C_VEL
LIN {X 0,Y 206.887,Z 158.68,A -85,B 0,C 180,E1 -23361.008,E2 -23361.008} C_VEL
LIN {X 0,Y 201.292,Z 147.947,A -85,B 0,C 180,E1 -23363.357,E2 -23363.357} C_VEL
LIN {X 0,Y 194.835,Z 137.17,A -85,B 0,C 180,E1 -23366.307,E2 -23366.307} C_VEL
LIN {X 0,Y 188.354,Z 127.328,A -85,B 0,C 180,E1 -23369.653,E2 -23369.653} C_VEL
LIN {X 0,Y 184.605,Z 122.336,A -85,B 0,C 180,E1 -23371.797,E2 -23371.797} C_VEL
LIN {X 0,Y 181.566,Z 118.221,A -85,B 0,C 180,E1 -23373.712,E2 -23373.712} C_VEL
LIN {X 0,Y 178.792,Z 114.704,A -85,B 0,C 180,E1 -23375.607,E2 -23375.607} C_VEL
LIN {X 0,Y 178.098,Z 113.643,A -85,B 0,C 180,E1 -23376.125,E2 -23376.125} C_VEL
LIN {X 0,Y 175.385,Z 110.823,A -85,B 0,C 180,E1 -23378.165,E2 -23378.165} C_VEL
LIN {X 0,Y 174.073,Z 108.511,A -85,B 0,C 180,E1 -23379.33,E2 -23379.33} C_VEL
LIN {X 0,Y 171.584,Z 106.504,A -85,B 0,C 180,E1 -23381.491,E2 -23381.491} C_VEL
LIN {X 0,Y 169.833,Z 103.37,A -85,B 0,C 180,E1 -23383.393,E2 -23383.393} C_VEL
LIN {X 0,Y 169.516,Z 102.91,A -85,B 0,C 180,E1 -23383.748,E2 -23383.748} C_VEL
LIN {X 0,Y 166.719,Z 101.265,A -85,B 0,C 180,E1 -23386.903,E2 -23386.903} C_VEL
LIN {X 0,Y 165.242,Z 98.842,A -85,B 0,C 180,E1 -23389.16,E2 -23389.16} C_VEL
LIN {X 0,Y 164.788,Z 96.953,A -85,B 0,C 180,E1 -23390.254,E2 -23390.254} C_VEL
LIN {X 0,Y 164.823,Z 96.936,A -85,B 0,C 180,E1 -23392.65,E2 -23392.65} C_VEL
LIN {X 0,Y 165.277,Z 96.874,A -85,B 0,C 180,E1 -23399.999,E2 -23399.999} C_VEL
LIN {X 0,Y 164.824,Z 96.936,A -85,B 0,C 180,E1 -23407.349,E2 -23407.349} C_VEL
LIN {X 0,Y 164.705,Z 96.947,A -85,B 0,C 180,E1 -23411.059,E2 -23411.059} C_VEL
LIN {X 0,Y 164.504,Z 97.17,A -85,B 0,C 180,E1 -23415.883,E2 -23415.883} C_VEL
LIN {X 0,Y 165.399,Z 99.679,A -85,B 0,C 180,E1 -23417.622,E2 -23417.622} C_VEL
LIN {X 0,Y 167.798,Z 102.188,A -85,B 0,C 180,E1 -23420.855,E2 -23420.855} C_VEL
LIN {X 0,Y 169.663,Z 103.2,A -85,B 0,C 180,E1 -23422.851,E2 -23422.851} C_VEL
LIN {X 0,Y 171.189,Z 106.131,A -85,B 0,C 180,E1 -23424.559,E2 -23424.559} C_VEL
LIN {X 0,Y 175.112,Z 110.437,A -85,B 0,C 180,E1 -23428.032,E2 -23428.032} C_VEL
LIN {X 0,Y 178.579,Z 115.694,A -85,B 0,C 180,E1 -23430.771,E2 -23430.771} C_VEL
LIN {X 0,Y 181.071,Z 119.579,A -85,B 0,C 180,E1 -23432.543,E2 -23432.543} C_VEL
LIN {X 0,Y 183.723,Z 123.597,A -85,B 0,C 180,E1 -23434.27,E2 -23434.27} C_VEL
LIN {X 0,Y 187.045,Z 129.024,A -85,B 0,C 180,E1 -23436.284,E2 -23436.284} C_VEL
LIN {X 0,Y 192.328,Z 138.318,A -85,B 0,C 180,E1 -23439.191,E2 -23439.191} C_VEL
LIN {X 0,Y 197.829,Z 149.1,A -85,B 0,C 180,E1 -23441.928,E2 -23441.928} C_VEL
LIN {X 0,Y 202.92,Z 160.8,A -85,B 0,C 180,E1 -23444.29,E2 -23444.29} C_VEL
LIN {X 0,Y 205.616,Z 167.934,A -85,B 0,C 180,E1 -23445.499,E2 -23445.499} C_VEL
LIN {X 0,Y 206.053,Z 172.886,A -85,B 0,C 180,E1 -23445.88,E2 -23445.88} C_VEL
LIN {X 0,Y 203.545,Z 209.378,A -85,B 0,C 180,E1 -23447.057,E2 -23447.057} C_VEL
LIN {X 0,Y 201.589,Z 222.844,A -85,B 0,C 180,E1 -23447.792,E2 -23447.792} C_VEL
LIN {X 0,Y 198.813,Z 235.551,A -85,B 0,C 180,E1 -23448.822,E2 -23448.822} C_VEL
LIN {X 0,Y 195.088,Z 248.124,A -85,B 0,C 180,E1 -23450.249,E2 -23450.249} C_VEL
LIN {X 0,Y 191.002,Z 259.335,A -85,B 0,C 180,E1 -23451.951,E2 -23451.951} C_VEL
LIN {X 0,Y 190.153,Z 261.657,A -85,B 0,C 180,E1 -23452.397,E2 -23452.397} C_VEL
LIN {X 0,Y 187.829,Z 266.364,A -85,B 0,C 180,E1 -23453.242,E2 -23453.242} C_VEL
LIN {X 0,Y 182.227,Z 273.607,A -85,B 0,C 180,E1 -23454.402,E2 -23454.402} C_VEL
LIN {X 0,Y 176.307,Z 280.351,A -85,B 0,C 180,E1 -23455.763,E2 -23455.763} C_VEL
LIN {X 0,Y 173.54,Z 284.173,A -85,B 0,C 180,E1 -23456.929,E2 -23456.929} C_VEL
LIN {X 0,Y 168.958,Z 291.81,A -85,B 0,C 180,E1 -23460.055,E2 -23460.055} C_VEL
LIN {X 0,Y 164.528,Z 298.878,A -85,B 0,C 180,E1 -23463.958,E2 -23463.958} C_VEL
LIN {X 0,Y 160.734,Z 304.504,A -85,B 0,C 180,E1 -23468.181,E2 -23468.181} C_VEL
LIN {X 0,Y 158.215,Z 308.038,A -85,B 0,C 180,E1 -23471.883,E2 -23471.883} C_VEL
LIN {X 0,Y 156.881,Z 309.836,A -85,B 0,C 180,E1 -23474.407,E2 -23474.407} C_VEL
LIN {X 0,Y 155.311,Z 312.212,A -85,B 0,C 180,E1 -23479.571,E2 -23479.571} C_VEL
LIN {X 0,Y 154.929,Z 312.823,A -85,B 0,C 180,E1 -23482.178,E2 -23482.178} C_VEL
LIN {X 0,Y 154.855,Z 312.905,A -85,B 0,C 180,E1 -23486.813,E2 -23486.813} C_VEL
LIN {X 0,Y 155.06,Z 312.203,A -85,B 0,C 180,E1 -23489.999,E2 -23489.999} C_VEL
LIN {X 0,Y 154.896,Z 310.745,A -85,B 0,C 180,E1 -23493.446,E2 -23493.446} C_VEL
LIN {X 0,Y 154.952,Z 307.798,A -85,B 0,C 180,E1 -23497.82,E2 -23497.82} C_VEL
LIN {X 0,Y 155.509,Z 304.069,A -85,B 0,C 180,E1 -23501.733,E2 -23501.733} C_VEL
LIN {X 0,Y 156.643,Z 299.203,A -85,B 0,C 180,E1 -23505.616,E2 -23505.616} C_VEL
LIN {X 0,Y 158.584,Z 293.072,A -85,B 0,C 180,E1 -23509.412,E2 -23509.412} C_VEL
LIN {X 0,Y 161.035,Z 285.429,A -85,B 0,C 180,E1 -23513.127,E2 -23513.127} C_VEL
LIN {X 0,Y 163.419,Z 277.596,A -85,B 0,C 180,E1 -23516.155,E2 -23516.155} C_VEL
LIN {X 0,Y 166.493,Z 268.051,A -85,B 0,C 180,E1 -23519.04,E2 -23519.04} C_VEL
LIN {X 0,Y 169.669,Z 257.464,A -85,B 0,C 180,E1 -23521.53,E2 -23521.53} C_VEL
LIN {X 0,Y 172.718,Z 245.65,A -85,B 0,C 180,E1 -23523.669,E2 -23523.669} C_VEL
LIN {X 0,Y 175.241,Z 234.135,A -85,B 0,C 180,E1 -23525.204,E2 -23525.204} C_VEL
LIN {X 0,Y 177.421,Z 220.566,A -85,B 0,C 180,E1 -23526.516,E2 -23526.516} C_VEL
LIN {X 0,Y 178.764,Z 207.743,A -85,B 0,C 180,E1 -23527.324,E2 -23527.324} C_VEL
LIN {X 0,Y 181.013,Z 164.181,A -85,B 0,C 180,E1 -23528.949,E2 -23528.949} C_VEL
LIN {X 0,Y 179.287,Z 144.176,A -85,B 0,C 180,E1 -23530.317,E2 -23530.317} C_VEL
LIN {X 0,Y 173.52,Z 129.235,A -85,B 0,C 180,E1 -23532.53,E2 -23532.53} C_VEL
LIN {X 0,Y 167.621,Z 116.991,A -85,B 0,C 180,E1 -23534.859,E2 -23534.859} C_VEL
LIN {X 0,Y 162.854,Z 108.213,A -85,B 0,C 180,E1 -23536.866,E2 -23536.866} C_VEL
LIN {X 0,Y 160.107,Z 103.505,A -85,B 0,C 180,E1 -23538.088,E2 -23538.088} C_VEL
LIN {X 0,Y 157.639,Z 99.542,A -85,B 0,C 180,E1 -23539.228,E2 -23539.228} C_VEL
LIN {X 0,Y 157.418,Z 98.861,A -85,B 0,C 180,E1 -23539.372,E2 -23539.372} C_VEL
LIN {X 0,Y 157.245,Z 97.865,A -85,B 0,C 180,E1 -23540.298,E2 -23540.298} C_VEL
LIN {X 0,Y 157.274,Z 97.887,A -85,B 0,C 180,E1 -23544.485,E2 -23544.485} C_VEL
LIN {X 0,Y 157.292,Z 97.892,A -85,B 0,C 180,E1 -23548.095,E2 -23548.095} C_VEL
LIN {X 0,Y 157.321,Z 97.875,A -85,B 0,C 180,E1 -23553.466,E2 -23553.466} C_VEL
LIN {X 0,Y 157.393,Z 97.86,A -85,B 0,C 180,E1 -23559.668,E2 -23559.668} C_VEL
LIN {X 0,Y 157.454,Z 97.869,A -85,B 0,C 180,E1 -23564.466,E2 -23564.466} C_VEL
LIN {X 0,Y 157.689,Z 97.831,A -85,B 0,C 180,E1 -23569.731,E2 -23569.731} C_VEL
LIN {X 0,Y 157.767,Z 97.833,A -85,B 0,C 180,E1 -23572.321,E2 -23572.321} C_VEL
LIN {X 0,Y 158.254,Z 97.771,A -85,B 0,C 180,E1 -23580.001,E2 -23580.001} C_VEL
LIN {X 0,Y 157.763,Z 97.827,A -85,B 0,C 180,E1 -23587.681,E2 -23587.681} C_VEL
LIN {X 0,Y 157.633,Z 97.834,A -85,B 0,C 180,E1 -23591.231,E2 -23591.231} C_VEL
LIN {X 0,Y 157.441,Z 97.863,A -85,B 0,C 180,E1 -23595.536,E2 -23595.536} C_VEL
LIN {X 0,Y 157.37,Z 97.859,A -85,B 0,C 180,E1 -23600.934,E2 -23600.934} C_VEL
LIN {X 0,Y 157.314,Z 97.885,A -85,B 0,C 180,E1 -23606.685,E2 -23606.685} C_VEL
LIN {X 0,Y 157.275,Z 97.894,A -85,B 0,C 180,E1 -23612.429,E2 -23612.429} C_VEL
LIN {X 0,Y 157.259,Z 97.898,A -85,B 0,C 180,E1 -23616.446,E2 -23616.446} C_VEL
LIN {X 0,Y 157.19,Z 97.904,A -85,B 0,C 180,E1 -23622.118,E2 -23622.118} C_VEL
LIN {X 0,Y 157.189,Z 97.903,A -85,B 0,C 180,E1 -23628.108,E2 -23628.108} C_VEL
LIN {X 0,Y 158.272,Z 100.891,A -85,B 0,C 180,E1 -23628.789,E2 -23628.789} C_VEL
LIN {X 0,Y 160.407,Z 103.261,A -85,B 0,C 180,E1 -23629.701,E2 -23629.701} C_VEL
LIN {X 0,Y 162.65,Z 106.706,A -85,B 0,C 180,E1 -23630.674,E2 -23630.674} C_VEL
LIN {X 0,Y 170.077,Z 118.174,A -85,B 0,C 180,E1 -23633.625,E2 -23633.625} C_VEL
LIN {X 0,Y 177.402,Z 131.678,A -85,B 0,C 180,E1 -23636.3,E2 -23636.3} C_VEL
LIN {X 0,Y 182.145,Z 141.955,A -85,B 0,C 180,E1 -23637.945,E2 -23637.945} C_VEL
LIN {X 0,Y 179.27,Z 195.465,A -85,B 0,C 180,E1 -23639.922,E2 -23639.922} C_VEL
LIN {X 0,Y 177.857,Z 209.133,A -85,B 0,C 180,E1 -23640.857,E2 -23640.857} C_VEL
LIN {X 0,Y 176.03,Z 221.809,A -85,B 0,C 180,E1 -23642.185,E2 -23642.185} C_VEL
LIN {X 0,Y 173.722,Z 233.662,A -85,B 0,C 180,E1 -23643.9,E2 -23643.9} C_VEL
LIN {X 0,Y 170.964,Z 245.028,A -85,B 0,C 180,E1 -23646.051,E2 -23646.051} C_VEL
LIN {X 0,Y 168.054,Z 255.286,A -85,B 0,C 180,E1 -23648.536,E2 -23648.536} C_VEL
LIN {X 0,Y 165.061,Z 264.514,A -85,B 0,C 180,E1 -23651.378,E2 -23651.378} C_VEL
LIN {X 0,Y 162.108,Z 273.445,A -85,B 0,C 180,E1 -23654.923,E2 -23654.923} C_VEL
LIN {X 0,Y 159.6,Z 280.652,A -85,B 0,C 180,E1 -23658.572,E2 -23658.572} C_VEL
LIN {X 0,Y 157.721,Z 286.417,A -85,B 0,C 180,E1 -23662.319,E2 -23662.319} C_VEL
LIN {X 0,Y 156.29,Z 290.965,A -85,B 0,C 180,E1 -23666.133,E2 -23666.133} C_VEL
LIN {X 0,Y 155.497,Z 294.426,A -85,B 0,C 180,E1 -23670.001,E2 -23670.001} C_VEL
LIN {X 0,Y 155.143,Z 297.285,A -85,B 0,C 180,E1 -23674.712,E2 -23674.712} C_VEL
LIN {X 0,Y 154.953,Z 298.454,A -85,B 0,C 180,E1 -23677.821,E2 -23677.821} C_VEL
LIN {X 0,Y 155.073,Z 299.015,A -85,B 0,C 180,E1 -23680.445,E2 -23680.445} C_VEL
LIN {X 0,Y 156.008,Z 298.881,A -85,B 0,C 180,E1 -23685.683,E2 -23685.683} C_VEL
LIN {X 0,Y 156.888,Z 298.231,A -85,B 0,C 180,E1 -23688.276,E2 -23688.276} C_VEL
LIN {X 0,Y 158.156,Z 297.059,A -85,B 0,C 180,E1 -23691.062,E2 -23691.062} C_VEL
LIN {X 0,Y 160.977,Z 293.747,A -85,B 0,C 180,E1 -23695.887,E2 -23695.887} C_VEL
LIN {X 0,Y 163.911,Z 289.982,A -85,B 0,C 180,E1 -23699.544,E2 -23699.544} C_VEL
LIN {X 0,Y 167.399,Z 285.066,A -85,B 0,C 180,E1 -23703.079,E2 -23703.079} C_VEL
LIN {X 0,Y 171.509,Z 278.845,A -85,B 0,C 180,E1 -23706.455,E2 -23706.455} C_VEL
LIN {X 0,Y 176.145,Z 271.026,A -85,B 0,C 180,E1 -23709.672,E2 -23709.672} C_VEL
LIN {X 0,Y 180.937,Z 261.561,A -85,B 0,C 180,E1 -23712.673,E2 -23712.673} C_VEL
LIN {X 0,Y 185.253,Z 252.086,A -85,B 0,C 180,E1 -23714.958,E2 -23714.958} C_VEL
LIN {X 0,Y 189.193,Z 242.152,A -85,B 0,C 180,E1 -23716.805,E2 -23716.805} C_VEL
LIN {X 0,Y 192.765,Z 231.302,A -85,B 0,C 180,E1 -23718.367,E2 -23718.367} C_VEL
LIN {X 0,Y 195.855,Z 218.842,A -85,B 0,C 180,E1 -23719.765,E2 -23719.765} C_VEL
LIN {X 0,Y 198.321,Z 206.358,A -85,B 0,C 180,E1 -23720.708,E2 -23720.708} C_VEL
LIN {X 0,Y 199.912,Z 192.691,A -85,B 0,C 180,E1 -23721.39,E2 -23721.39} C_VEL
LIN {X 0,Y 202.001,Z 161.384,A -85,B 0,C 180,E1 -23722.4,E2 -23722.4} C_VEL
LIN {X 0,Y 195.823,Z 149.702,A -85,B 0,C 180,E1 -23725.193,E2 -23725.193} C_VEL
LIN {X 0,Y 189.714,Z 139.608,A -85,B 0,C 180,E1 -23728.243,E2 -23728.243} C_VEL
LIN {X 0,Y 184.876,Z 132.361,A -85,B 0,C 180,E1 -23730.942,E2 -23730.942} C_VEL
LIN {X 0,Y 181.983,Z 128.259,A -85,B 0,C 180,E1 -23732.712,E2 -23732.712} C_VEL
LIN {X 0,Y 179.094,Z 124.274,A -85,B 0,C 180,E1 -23734.631,E2 -23734.631} C_VEL
LIN {X 0,Y 176.308,Z 120.498,A -85,B 0,C 180,E1 -23736.66,E2 -23736.66} C_VEL
LIN {X 0,Y 173.021,Z 116.569,A -85,B 0,C 180,E1 -23739.305,E2 -23739.305} C_VEL
LIN {X 0,Y 172.106,Z 115.079,A -85,B 0,C 180,E1 -23740.152,E2 -23740.152} C_VEL
LIN {X 0,Y 169.58,Z 112.666,A -85,B 0,C 180,E1 -23742.514,E2 -23742.514} C_VEL
LIN {X 0,Y 167.841,Z 109.71,A -85,B 0,C 180,E1 -23744.517,E2 -23744.517} C_VEL
LIN {X 0,Y 165.198,Z 107.846,A -85,B 0,C 180,E1 -23747.718,E2 -23747.718} C_VEL
LIN {X 0,Y 163.733,Z 105.11,A -85,B 0,C 180,E1 -23750.191,E2 -23750.191} C_VEL
LIN {X 0,Y 163.349,Z 103.906,A -85,B 0,C 180,E1 -23751.027,E2 -23751.027} C_VEL
LIN {X 0,Y 160.352,Z 102.184,A -85,B 0,C 180,E1 -23758.744,E2 -23758.744} C_VEL
LIN {X 0,Y 160.164,Z 101.772,A -85,B 0,C 180,E1 -23759.999,E2 -23759.999} C_VEL
LIN {X 0,Y 160.572,Z 102.681,A -85,B 0,C 180,E1 -23768.811,E2 -23768.811} C_VEL
LIN {X 0,Y 163.208,Z 104.122,A -85,B 0,C 180,E1 -23775.212,E2 -23775.212} C_VEL
LIN {X 0,Y 164.419,Z 106.958,A -85,B 0,C 180,E1 -23777.549,E2 -23777.549} C_VEL
LIN {X 0,Y 166.913,Z 109.293,A -85,B 0,C 180,E1 -23780.89,E2 -23780.89} C_VEL
LIN {X 0,Y 168.015,Z 109.981,A -85,B 0,C 180,E1 -23782.115,E2 -23782.115} C_VEL
LIN {X 0,Y 169.915,Z 113.224,A -85,B 0,C 180,E1 -23784.269,E2 -23784.269} C_VEL
LIN {X 0,Y 173.068,Z 116.82,A -85,B 0,C 180,E1 -23787.18,E2 -23787.18} C_VEL
LIN {X 0,Y 177.458,Z 123.662,A -85,B 0,C 180,E1 -23790.764,E2 -23790.764} C_VEL
LIN {X 0,Y 181.168,Z 129.628,A -85,B 0,C 180,E1 -23793.38,E2 -23793.38} C_VEL
LIN {X 0,Y 184.144,Z 134.67,A -85,B 0,C 180,E1 -23795.289,E2 -23795.289} C_VEL
LIN {X 0,Y 189.014,Z 143.53,A -85,B 0,C 180,E1 -23798.135,E2 -23798.135} C_VEL
LIN {X 0,Y 194.345,Z 154.378,A -85,B 0,C 180,E1 -23800.952,E2 -23800.952} C_VEL
LIN {X 0,Y 198.981,Z 165.485,A -85,B 0,C 180,E1 -23803.243,E2 -23803.243} C_VEL
LIN {X 0,Y 201.011,Z 171.342,A -85,B 0,C 180,E1 -23804.232,E2 -23804.232} C_VEL
LIN {X 0,Y 201.151,Z 175.035,A -85,B 0,C 180,E1 -23804.473,E2 -23804.473} C_VEL
LIN {X 0,Y 198.672,Z 209.257,A -85,B 0,C 180,E1 -23805.589,E2 -23805.589} C_VEL
LIN {X 0,Y 196.702,Z 222.361,A -85,B 0,C 180,E1 -23806.308,E2 -23806.308} C_VEL
LIN {X 0,Y 194.103,Z 234.051,A -85,B 0,C 180,E1 -23807.242,E2 -23807.242} C_VEL
LIN {X 0,Y 190.778,Z 245.358,A -85,B 0,C 180,E1 -23808.463,E2 -23808.463} C_VEL
LIN {X 0,Y 186.488,Z 257.021,A -85,B 0,C 180,E1 -23810.158,E2 -23810.158} C_VEL
LIN {X 0,Y 182.114,Z 267.507,A -85,B 0,C 180,E1 -23812.219,E2 -23812.219} C_VEL
LIN {X 0,Y 177.949,Z 276.094,A -85,B 0,C 180,E1 -23814.369,E2 -23814.369} C_VEL
LIN {X 0,Y 173.54,Z 284.173,A -85,B 0,C 180,E1 -23816.929,E2 -23816.929} C_VEL
LIN {X 0,Y 170.814,Z 287.842,A -85,B 0,C 180,E1 -23818.203,E2 -23818.203} C_VEL
LIN {X 0,Y 164.925,Z 293.286,A -85,B 0,C 180,E1 -23820.197,E2 -23820.197} C_VEL
LIN {X 0,Y 159.217,Z 298.108,A -85,B 0,C 180,E1 -23822.484,E2 -23822.484} C_VEL
LIN {X 0,Y 156.839,Z 300.689,A -85,B 0,C 180,E1 -23824.192,E2 -23824.192} C_VEL
LIN {X 0,Y 153.184,Z 305.592,A -85,B 0,C 180,E1 -23828.466,E2 -23828.466} C_VEL
LIN {X 0,Y 151.447,Z 307.832,A -85,B 0,C 180,E1 -23831.043,E2 -23831.043} C_VEL
LIN {X 0,Y 150.018,Z 309.596,A -85,B 0,C 180,E1 -23833.674,E2 -23833.674} C_VEL
LIN {X 0,Y 148.305,Z 311.935,A -85,B 0,C 180,E1 -23839.072,E2 -23839.072} C_VEL
LIN {X 0,Y 147.876,Z 312.525,A -85,B 0,C 180,E1 -23841.802,E2 -23841.802} C_VEL
LIN {X 0,Y 147.79,Z 312.503,A -85,B 0,C 180,E1 -23846.998,E2 -23846.998} C_VEL
LIN {X 0,Y 147.963,Z 311.837,A -85,B 0,C 180,E1 -23849.999,E2 -23849.999} C_VEL
LIN {X 0,Y 147.813,Z 310.578,A -85,B 0,C 180,E1 -23853.169,E2 -23853.169} C_VEL
LIN {X 0,Y 147.894,Z 307.355,A -85,B 0,C 180,E1 -23858.195,E2 -23858.195} C_VEL
LIN {X 0,Y 148.526,Z 303.584,A -85,B 0,C 180,E1 -23862.293,E2 -23862.293} C_VEL
LIN {X 0,Y 149.777,Z 298.674,A -85,B 0,C 180,E1 -23866.351,E2 -23866.351} C_VEL
LIN {X 0,Y 151.826,Z 292.491,A -85,B 0,C 180,E1 -23870.314,E2 -23870.314} C_VEL
LIN {X 0,Y 154.049,Z 286.172,A -85,B 0,C 180,E1 -23873.527,E2 -23873.527} C_VEL
LIN {X 0,Y 157.014,Z 276.876,A -85,B 0,C 180,E1 -23877.308,E2 -23877.308} C_VEL
LIN {X 0,Y 160.302,Z 267.242,A -85,B 0,C 180,E1 -23880.276,E2 -23880.276} C_VEL
LIN {X 0,Y 163.658,Z 256.555,A -85,B 0,C 180,E1 -23882.83,E2 -23882.83} C_VEL
LIN {X 0,Y 166.416,Z 246.217,A -85,B 0,C 180,E1 -23884.758,E2 -23884.758} C_VEL
LIN {X 0,Y 169.238,Z 233.915,A -85,B 0,C 180,E1 -23886.466,E2 -23886.466} C_VEL
LIN {X 0,Y 171.441,Z 220.93,A -85,B 0,C 180,E1 -23887.758,E2 -23887.758} C_VEL
LIN {X 0,Y 172.88,Z 208.212,A -85,B 0,C 180,E1 -23888.601,E2 -23888.601} C_VEL
LIN {X 0,Y 175.226,Z 164.398,A -85,B 0,C 180,E1 -23890.294,E2 -23890.294} C_VEL
LIN {X 0,Y 173.716,Z 146.532,A -85,B 0,C 180,E1 -23891.581,E2 -23891.581} C_VEL
LIN {X 0,Y 168.295,Z 132.276,A -85,B 0,C 180,E1 -23893.815,E2 -23893.815} C_VEL
LIN {X 0,Y 162.863,Z 120.896,A -85,B 0,C 180,E1 -23896.114,E2 -23896.114} C_VEL
LIN {X 0,Y 157.875,Z 111.666,A -85,B 0,C 180,E1 -23898.373,E2 -23898.373} C_VEL
LIN {X 0,Y 155.954,Z 108.299,A -85,B 0,C 180,E1 -23899.295,E2 -23899.295} C_VEL
LIN {X 0,Y 153.184,Z 103.691,A -85,B 0,C 180,E1 -23900.676,E2 -23900.676} C_VEL
LIN {X 0,Y 151.03,Z 101.392,A -85,B 0,C 180,E1 -23901.722,E2 -23901.722} C_VEL
LIN {X 0,Y 150.169,Z 98.745,A -85,B 0,C 180,E1 -23902.315,E2 -23902.315} C_VEL
LIN {X 0,Y 150.214,Z 98.773,A -85,B 0,C 180,E1 -23907.368,E2 -23907.368} C_VEL
LIN {X 0,Y 150.243,Z 98.757,A -85,B 0,C 180,E1 -23912.718,E2 -23912.718} C_VEL
LIN {X 0,Y 150.35,Z 98.738,A -85,B 0,C 180,E1 -23919.208,E2 -23919.208} C_VEL
LIN {X 0,Y 150.362,Z 98.755,A -85,B 0,C 180,E1 -23923.714,E2 -23923.714} C_VEL
LIN {X 0,Y 150.61,Z 98.707,A -85,B 0,C 180,E1 -23929.243,E2 -23929.243} C_VEL
LIN {X 0,Y 150.704,Z 98.713,A -85,B 0,C 180,E1 -23931.958,E2 -23931.958} C_VEL
LIN {X 0,Y 151.215,Z 98.648,A -85,B 0,C 180,E1 -23940.001,E2 -23940.001} C_VEL
LIN {X 0,Y 150.701,Z 98.708,A -85,B 0,C 180,E1 -23948.043,E2 -23948.043} C_VEL
LIN {X 0,Y 150.575,Z 98.711,A -85,B 0,C 180,E1 -23951.434,E2 -23951.434} C_VEL
LIN {X 0,Y 150.353,Z 98.751,A -85,B 0,C 180,E1 -23956.288,E2 -23956.288} C_VEL
LIN {X 0,Y 150.351,Z 98.733,A -85,B 0,C 180,E1 -23960.793,E2 -23960.793} C_VEL
LIN {X 0,Y 150.244,Z 98.764,A -85,B 0,C 180,E1 -23967.283,E2 -23967.283} C_VEL
LIN {X 0,Y 150.214,Z 98.774,A -85,B 0,C 180,E1 -23972.633,E2 -23972.633} C_VEL
LIN {X 0,Y 150.169,Z 98.778,A -85,B 0,C 180,E1 -23977.476,E2 -23977.476} C_VEL
LIN {X 0,Y 150.133,Z 98.781,A -85,B 0,C 180,E1 -23981.498,E2 -23981.498} C_VEL
LIN {X 0,Y 150.13,Z 98.784,A -85,B 0,C 180,E1 -23985.398,E2 -23985.398} C_VEL
LIN {X 0,Y 151.098,Z 101.573,A -85,B 0,C 180,E1 -23986.017,E2 -23986.017} C_VEL
LIN {X 0,Y 153.18,Z 103.784,A -85,B 0,C 180,E1 -23987.027,E2 -23987.027} C_VEL
LIN {X 0,Y 155.567,Z 107.522,A -85,B 0,C 180,E1 -23988.207,E2 -23988.207} C_VEL
LIN {X 0,Y 156.964,Z 109.388,A -85,B 0,C 180,E1 -23988.849,E2 -23988.849} C_VEL
LIN {X 0,Y 162.415,Z 117.624,A -85,B 0,C 180,E1 -23991.246,E2 -23991.246} C_VEL
LIN {X 0,Y 167.893,Z 126.811,A -85,B 0,C 180,E1 -23993.466,E2 -23993.466} C_VEL
LIN {X 0,Y 174.018,Z 138.762,A -85,B 0,C 180,E1 -23995.796,E2 -23995.796} C_VEL
LIN {X 0,Y 176.362,Z 144.154,A -85,B 0,C 180,E1 -23996.668,E2 -23996.668} C_VEL
LIN {X 0,Y 173.405,Z 196.101,A -85,B 0,C 180,E1 -23998.634,E2 -23998.634} C_VEL
LIN {X 0,Y 171.977,Z 209.411,A -85,B 0,C 180,E1 -23999.572,E2 -23999.572} C_VEL
LIN {X 0,Y 170.033,Z 222.208,A -85,B 0,C 180,E1 -24000.945,E2 -24000.945} C_VEL
LIN {X 0,Y 167.806,Z 233.254,A -85,B 0,C 180,E1 -24002.569,E2 -24002.569} C_VEL
LIN {X 0,Y 164.913,Z 244.752,A -85,B 0,C 180,E1 -24004.776,E2 -24004.776} C_VEL
LIN {X 0,Y 161.832,Z 255.115,A -85,B 0,C 180,E1 -24007.331,E2 -24007.331} C_VEL
LIN {X 0,Y 158.981,Z 263.597,A -85,B 0,C 180,E1 -24009.965,E2 -24009.965} C_VEL
LIN {X 0,Y 156.249,Z 271.413,A -85,B 0,C 180,E1 -24013.001,E2 -24013.001} C_VEL
LIN {X 0,Y 153.489,Z 279.049,A -85,B 0,C 180,E1 -24016.766,E2 -24016.766} C_VEL
LIN {X 0,Y 151.326,Z 285.181,A -85,B 0,C 180,E1 -24020.646,E2 -24020.646} C_VEL
LIN {X 0,Y 149.645,Z 290.062,A -85,B 0,C 180,E1 -24024.611,E2 -24024.611} C_VEL
LIN {X 0,Y 148.615,Z 293.828,A -85,B 0,C 180,E1 -24028.646,E2 -24028.646} C_VEL
LIN {X 0,Y 148.08,Z 296.588,A -85,B 0,C 180,E1 -24032.721,E2 -24032.721} C_VEL
LIN {X 0,Y 147.946,Z 297.899,A -85,B 0,C 180,E1 -24035.453,E2 -24035.453} C_VEL
LIN {X 0,Y 147.867,Z 298.831,A -85,B 0,C 180,E1 -24038.198,E2 -24038.198} C_VEL
LIN {X 0,Y 148.017,Z 299.356,A -85,B 0,C 180,E1 -24040.949,E2 -24040.949} C_VEL
LIN {X 0,Y 149.093,Z 299.173,A -85,B 0,C 180,E1 -24046.43,E2 -24046.43} C_VEL
LIN {X 0,Y 151.281,Z 297.469,A -85,B 0,C 180,E1 -24051.698,E2 -24051.698} C_VEL
LIN {X 0,Y 152.768,Z 295.878,A -85,B 0,C 180,E1 -24054.46,E2 -24054.46} C_VEL
LIN {X 0,Y 155.49,Z 292.775,A -85,B 0,C 180,E1 -24058.334,E2 -24058.334} C_VEL
LIN {X 0,Y 158.831,Z 288.587,A -85,B 0,C 180,E1 -24062.072,E2 -24062.072} C_VEL
LIN {X 0,Y 163.522,Z 282.18,A -85,B 0,C 180,E1 -24066.226,E2 -24066.226} C_VEL
LIN {X 0,Y 168.137,Z 275.13,A -85,B 0,C 180,E1 -24069.602,E2 -24069.602} C_VEL
LIN {X 0,Y 173.206,Z 266.306,A -85,B 0,C 180,E1 -24072.799,E2 -24072.799} C_VEL
LIN {X 0,Y 177.733,Z 257.147,A -85,B 0,C 180,E1 -24075.38,E2 -24075.38} C_VEL
LIN {X 0,Y 182.258,Z 247.024,A -85,B 0,C 180,E1 -24077.518,E2 -24077.518} C_VEL
LIN {X 0,Y 186.453,Z 235.714,A -85,B 0,C 180,E1 -24079.34,E2 -24079.34} C_VEL
LIN {X 0,Y 189.891,Z 223.96,A -85,B 0,C 180,E1 -24080.798,E2 -24080.798} C_VEL
LIN {X 0,Y 192.446,Z 212.629,A -85,B 0,C 180,E1 -24081.837,E2 -24081.837} C_VEL
LIN {X 0,Y 194.546,Z 199.613,A -85,B 0,C 180,E1 -24082.633,E2 -24082.633} C_VEL
LIN {X 0,Y 196.012,Z 182.129,A -85,B 0,C 180,E1 -24083.281,E2 -24083.281} C_VEL
LIN {X 0,Y 197.219,Z 164.262,A -85,B 0,C 180,E1 -24083.859,E2 -24083.859} C_VEL
LIN {X 0,Y 192.043,Z 154.359,A -85,B 0,C 180,E1 -24086.362,E2 -24086.362} C_VEL
LIN {X 0,Y 186.562,Z 145.027,A -85,B 0,C 180,E1 -24089.274,E2 -24089.274} C_VEL
LIN {X 0,Y 182.063,Z 138.069,A -85,B 0,C 180,E1 -24091.935,E2 -24091.935} C_VEL
LIN {X 0,Y 179.264,Z 134.003,A -85,B 0,C 180,E1 -24093.75,E2 -24093.75} C_VEL
LIN {X 0,Y 176.634,Z 130.272,A -85,B 0,C 180,E1 -24095.602,E2 -24095.602} C_VEL
LIN {X 0,Y 173.544,Z 126.099,A -85,B 0,C 180,E1 -24098,E2 -24098} C_VEL
LIN {X 0,Y 170.72,Z 122.35,A -85,B 0,C 180,E1 -24100.477,E2 -24100.477} C_VEL
LIN {X 0,Y 170.003,Z 121.445,A -85,B 0,C 180,E1 -24101.157,E2 -24101.157} C_VEL
LIN {X 0,Y 167.51,Z 118.611,A -85,B 0,C 180,E1 -24103.705,E2 -24103.705} C_VEL
LIN {X 0,Y 166.465,Z 116.566,A -85,B 0,C 180,E1 -24105.013,E2 -24105.013} C_VEL
LIN {X 0,Y 163.815,Z 114.53,A -85,B 0,C 180,E1 -24108.398,E2 -24108.398} C_VEL
LIN {X 0,Y 162.361,Z 111.644,A -85,B 0,C 180,E1 -24111.05,E2 -24111.05} C_VEL
LIN {X 0,Y 161.967,Z 110.817,A -85,B 0,C 180,E1 -24111.892,E2 -24111.892} C_VEL
LIN {X 0,Y 159.327,Z 108.987,A -85,B 0,C 180,E1 -24119.684,E2 -24119.684} C_VEL
LIN {X 0,Y 159.218,Z 109.34,A -85,B 0,C 180,E1 -24126.335,E2 -24126.335} C_VEL
LIN {X 0,Y 161.976,Z 111.084,A -85,B 0,C 180,E1 -24134.607,E2 -24134.607} C_VEL
LIN {X 0,Y 163.29,Z 113.928,A -85,B 0,C 180,E1 -24137.211,E2 -24137.211} C_VEL
LIN {X 0,Y 165.776,Z 116.261,A -85,B 0,C 180,E1 -24140.634,E2 -24140.634} C_VEL
LIN {X 0,Y 166.514,Z 116.929,A -85,B 0,C 180,E1 -24141.51,E2 -24141.51} C_VEL
LIN {X 0,Y 168.799,Z 120.413,A -85,B 0,C 180,E1 -24144.122,E2 -24144.122} C_VEL
LIN {X 0,Y 171.341,Z 123.679,A -85,B 0,C 180,E1 -24146.573,E2 -24146.573} C_VEL
LIN {X 0,Y 175.031,Z 129.558,A -85,B 0,C 180,E1 -24149.746,E2 -24149.746} C_VEL
LIN {X 0,Y 178.403,Z 135.208,A -85,B 0,C 180,E1 -24152.283,E2 -24152.283} C_VEL
LIN {X 0,Y 181.626,Z 140.96,A -85,B 0,C 180,E1 -24154.48,E2 -24154.48} C_VEL
LIN {X 0,Y 185.922,Z 149.03,A -85,B 0,C 180,E1 -24157.13,E2 -24157.13} C_VEL
LIN {X 0,Y 190.887,Z 159.615,A -85,B 0,C 180,E1 -24159.925,E2 -24159.925} C_VEL
LIN {X 0,Y 195.642,Z 171.501,A -85,B 0,C 180,E1 -24162.417,E2 -24162.417} C_VEL
LIN {X 0,Y 196.469,Z 174.267,A -85,B 0,C 180,E1 -24162.865,E2 -24162.865} C_VEL
LIN {X 0,Y 194.516,Z 203.248,A -85,B 0,C 180,E1 -24163.819,E2 -24163.819} C_VEL
LIN {X 0,Y 192.816,Z 216.808,A -85,B 0,C 180,E1 -24164.417,E2 -24164.417} C_VEL
LIN {X 0,Y 190.456,Z 228.764,A -85,B 0,C 180,E1 -24165.246,E2 -24165.246} C_VEL
LIN {X 0,Y 187.24,Z 240.58,A -85,B 0,C 180,E1 -24166.393,E2 -24166.393} C_VEL
LIN {X 0,Y 183.366,Z 251.854,A -85,B 0,C 180,E1 -24167.875,E2 -24167.875} C_VEL
LIN {X 0,Y 179.068,Z 262.168,A -85,B 0,C 180,E1 -24169.639,E2 -24169.639} C_VEL
LIN {X 0,Y 174.146,Z 272.602,A -85,B 0,C 180,E1 -24172.015,E2 -24172.015} C_VEL
LIN {X 0,Y 169.471,Z 281.066,A -85,B 0,C 180,E1 -24174.507,E2 -24174.507} C_VEL
LIN {X 0,Y 164.401,Z 289.339,A -85,B 0,C 180,E1 -24177.698,E2 -24177.698} C_VEL
LIN {X 0,Y 160.042,Z 296.029,A -85,B 0,C 180,E1 -24181.114,E2 -24181.114} C_VEL
LIN {X 0,Y 156.839,Z 300.689,A -85,B 0,C 180,E1 -24184.192,E2 -24184.192} C_VEL
LIN {X 0,Y 154.529,Z 303.075,A -85,B 0,C 180,E1 -24185.998,E2 -24185.998} C_VEL
LIN {X 0,Y 149.213,Z 306.356,A -85,B 0,C 180,E1 -24188.913,E2 -24188.913} C_VEL
LIN {X 0,Y 144.255,Z 308.914,A -85,B 0,C 180,E1 -24192.123,E2 -24192.123} C_VEL
LIN {X 0,Y 142.579,Z 310.058,A -85,B 0,C 180,E1 -24194.333,E2 -24194.333} C_VEL
LIN {X 0,Y 141.321,Z 311.659,A -85,B 0,C 180,E1 -24198.525,E2 -24198.525} C_VEL
LIN {X 0,Y 140.824,Z 312.22,A -85,B 0,C 180,E1 -24201.389,E2 -24201.389} C_VEL
LIN {X 0,Y 140.702,Z 312.11,A -85,B 0,C 180,E1 -24207.136,E2 -24207.136} C_VEL
LIN {X 0,Y 140.869,Z 311.471,A -85,B 0,C 180,E1 -24209.999,E2 -24209.999} C_VEL
LIN {X 0,Y 140.735,Z 310.407,A -85,B 0,C 180,E1 -24212.862,E2 -24212.862} C_VEL
LIN {X 0,Y 140.678,Z 308.874,A -85,B 0,C 180,E1 -24215.733,E2 -24215.733} C_VEL
LIN {X 0,Y 141.033,Z 305.773,A -85,B 0,C 180,E1 -24220.044,E2 -24220.044} C_VEL
LIN {X 0,Y 141.927,Z 301.59,A -85,B 0,C 180,E1 -24224.334,E2 -24224.334} C_VEL
LIN {X 0,Y 144.001,Z 295.206,A -85,B 0,C 180,E1 -24229.234,E2 -24229.234} C_VEL
LIN {X 0,Y 146.586,Z 288.254,A -85,B 0,C 180,E1 -24233.299,E2 -24233.299} C_VEL
LIN {X 0,Y 148.902,Z 281.423,A -85,B 0,C 180,E1 -24236.488,E2 -24236.488} C_VEL
LIN {X 0,Y 152.001,Z 272.519,A -85,B 0,C 180,E1 -24239.804,E2 -24239.804} C_VEL
LIN {X 0,Y 155.685,Z 261.915,A -85,B 0,C 180,E1 -24242.799,E2 -24242.799} C_VEL
LIN {X 0,Y 158.887,Z 251.398,A -85,B 0,C 180,E1 -24245.101,E2 -24245.101} C_VEL
LIN {X 0,Y 161.924,Z 239.816,A -85,B 0,C 180,E1 -24247.028,E2 -24247.028} C_VEL
LIN {X 0,Y 164.489,Z 227.79,A -85,B 0,C 180,E1 -24248.476,E2 -24248.476} C_VEL
LIN {X 0,Y 166.439,Z 214.592,A -85,B 0,C 180,E1 -24249.607,E2 -24249.607} C_VEL
LIN {X 0,Y 167.588,Z 201.199,A -85,B 0,C 180,E1 -24250.311,E2 -24250.311} C_VEL
LIN {X 0,Y 169.563,Z 165.213,A -85,B 0,C 180,E1 -24251.693,E2 -24251.693} C_VEL
LIN {X 0,Y 168.276,Z 149.001,A -85,B 0,C 180,E1 -24252.91,E2 -24252.91} C_VEL
LIN {X 0,Y 163.342,Z 135.897,A -85,B 0,C 180,E1 -24255.091,E2 -24255.091} C_VEL
LIN {X 0,Y 158.621,Z 125.615,A -85,B 0,C 180,E1 -24257.244,E2 -24257.244} C_VEL
LIN {X 0,Y 152.509,Z 113.959,A -85,B 0,C 180,E1 -24260.254,E2 -24260.254} C_VEL
LIN {X 0,Y 149.402,Z 109.115,A -85,B 0,C 180,E1 -24261.873,E2 -24261.873} C_VEL
LIN {X 0,Y 147.06,Z 106.011,A -85,B 0,C 180,E1 -24263.133,E2 -24263.133} C_VEL
LIN {X 0,Y 146.543,Z 104.848,A -85,B 0,C 180,E1 -24263.457,E2 -24263.457} C_VEL
LIN {X 0,Y 144.386,Z 102.937,A -85,B 0,C 180,E1 -24264.627,E2 -24264.627} C_VEL
LIN {X 0,Y 143.239,Z 100.324,A -85,B 0,C 180,E1 -24265.403,E2 -24265.403} C_VEL
LIN {X 0,Y 143.134,Z 99.655,A -85,B 0,C 180,E1 -24265.556,E2 -24265.556} C_VEL
LIN {X 0,Y 143.121,Z 99.658,A -85,B 0,C 180,E1 -24270.591,E2 -24270.591} C_VEL
LIN {X 0,Y 143.158,Z 99.638,A -85,B 0,C 180,E1 -24273.78,E2 -24273.78} C_VEL
LIN {X 0,Y 143.306,Z 99.613,A -85,B 0,C 180,E1 -24279.923,E2 -24279.923} C_VEL
LIN {X 0,Y 143.358,Z 99.611,A -85,B 0,C 180,E1 -24285.812,E2 -24285.812} C_VEL
LIN {X 0,Y 143.536,Z 99.583,A -85,B 0,C 180,E1 -24288.706,E2 -24288.706} C_VEL
LIN {X 0,Y 143.625,Z 99.594,A -85,B 0,C 180,E1 -24291.559,E2 -24291.559} C_VEL
LIN {X 0,Y 144.173,Z 99.525,A -85,B 0,C 180,E1 -24300.001,E2 -24300.001} C_VEL
LIN {X 0,Y 143.622,Z 99.592,A -85,B 0,C 180,E1 -24308.442,E2 -24308.442} C_VEL
LIN {X 0,Y 143.501,Z 99.589,A -85,B 0,C 180,E1 -24311.624,E2 -24311.624} C_VEL
LIN {X 0,Y 143.296,Z 99.632,A -85,B 0,C 180,E1 -24317.115,E2 -24317.115} C_VEL
LIN {X 0,Y 143.277,Z 99.612,A -85,B 0,C 180,E1 -24321.255,E2 -24321.255} C_VEL
LIN {X 0,Y 143.19,Z 99.644,A -85,B 0,C 180,E1 -24327.938,E2 -24327.938} C_VEL
LIN {X 0,Y 143.142,Z 99.654,A -85,B 0,C 180,E1 -24333.42,E2 -24333.42} C_VEL
LIN {X 0,Y 143.052,Z 99.668,A -85,B 0,C 180,E1 -24339.694,E2 -24339.694} C_VEL
LIN {X 0,Y 143.069,Z 99.662,A -85,B 0,C 180,E1 -24342.124,E2 -24342.124} C_VEL
LIN {X 0,Y 143.969,Z 102.402,A -85,B 0,C 180,E1 -24342.824,E2 -24342.824} C_VEL
LIN {X 0,Y 146.063,Z 104.6,A -85,B 0,C 180,E1 -24344.001,E2 -24344.001} C_VEL
LIN {X 0,Y 146.827,Z 105.61,A -85,B 0,C 180,E1 -24344.43,E2 -24344.43} C_VEL
LIN {X 0,Y 149.006,Z 108.829,A -85,B 0,C 180,E1 -24345.635,E2 -24345.635} C_VEL
LIN {X 0,Y 150.153,Z 110.29,A -85,B 0,C 180,E1 -24346.228,E2 -24346.228} C_VEL
LIN {X 0,Y 155.466,Z 118.049,A -85,B 0,C 180,E1 -24348.85,E2 -24348.85} C_VEL
LIN {X 0,Y 161.712,Z 128.225,A -85,B 0,C 180,E1 -24351.643,E2 -24351.643} C_VEL
LIN {X 0,Y 168.102,Z 140.536,A -85,B 0,C 180,E1 -24354.281,E2 -24354.281} C_VEL
LIN {X 0,Y 170.624,Z 146.144,A -85,B 0,C 180,E1 -24355.281,E2 -24355.281} C_VEL
LIN {X 0,Y 167.623,Z 196.683,A -85,B 0,C 180,E1 -24357.249,E2 -24357.249} C_VEL
LIN {X 0,Y 166.073,Z 210.309,A -85,B 0,C 180,E1 -24358.244,E2 -24358.244} C_VEL
LIN {X 0,Y 164.115,Z 222.609,A -85,B 0,C 180,E1 -24359.613,E2 -24359.613} C_VEL
LIN {X 0,Y 161.589,Z 234.417,A -85,B 0,C 180,E1 -24361.418,E2 -24361.418} C_VEL
LIN {X 0,Y 158.551,Z 245.763,A -85,B 0,C 180,E1 -24363.688,E2 -24363.688} C_VEL
LIN {X 0,Y 155.345,Z 256.004,A -85,B 0,C 180,E1 -24366.328,E2 -24366.328} C_VEL
LIN {X 0,Y 152.37,Z 264.388,A -85,B 0,C 180,E1 -24369.056,E2 -24369.056} C_VEL
LIN {X 0,Y 148.986,Z 273.465,A -85,B 0,C 180,E1 -24372.854,E2 -24372.854} C_VEL
LIN {X 0,Y 146.198,Z 280.776,A -85,B 0,C 180,E1 -24376.801,E2 -24376.801} C_VEL
LIN {X 0,Y 143.685,Z 287.501,A -85,B 0,C 180,E1 -24381.563,E2 -24381.563} C_VEL
LIN {X 0,Y 142.153,Z 291.945,A -85,B 0,C 180,E1 -24385.748,E2 -24385.748} C_VEL
LIN {X 0,Y 141.297,Z 295.322,A -85,B 0,C 180,E1 -24390.001,E2 -24390.001} C_VEL
LIN {X 0,Y 140.99,Z 297.792,A -85,B 0,C 180,E1 -24394.465,E2 -24394.465} C_VEL
LIN {X 0,Y 140.786,Z 299.208,A -85,B 0,C 180,E1 -24398.614,E2 -24398.614} C_VEL
LIN {X 0,Y 140.988,Z 299.69,A -85,B 0,C 180,E1 -24401.502,E2 -24401.502} C_VEL
LIN {X 0,Y 142.214,Z 299.465,A -85,B 0,C 180,E1 -24407.249,E2 -24407.249} C_VEL
LIN {X 0,Y 144.44,Z 297.865,A -85,B 0,C 180,E1 -24412.408,E2 -24412.408} C_VEL
LIN {X 0,Y 146.234,Z 296.081,A -85,B 0,C 180,E1 -24415.63,E2 -24415.63} C_VEL
LIN {X 0,Y 149.185,Z 292.931,A -85,B 0,C 180,E1 -24419.647,E2 -24419.647} C_VEL
LIN {X 0,Y 152.744,Z 288.693,A -85,B 0,C 180,E1 -24423.515,E2 -24423.515} C_VEL
LIN {X 0,Y 157.763,Z 282.23,A -85,B 0,C 180,E1 -24427.774,E2 -24427.774} C_VEL
LIN {X 0,Y 162.656,Z 275.089,A -85,B 0,C 180,E1 -24431.219,E2 -24431.219} C_VEL
LIN {X 0,Y 167.473,Z 267.091,A -85,B 0,C 180,E1 -24434.181,E2 -24434.181} C_VEL
LIN {X 0,Y 171.789,Z 258.914,A -85,B 0,C 180,E1 -24436.567,E2 -24436.567} C_VEL
LIN {X 0,Y 176.419,Z 249.131,A -85,B 0,C 180,E1 -24438.758,E2 -24438.758} C_VEL
LIN {X 0,Y 180.733,Z 238.367,A -85,B 0,C 180,E1 -24440.613,E2 -24440.613} C_VEL
LIN {X 0,Y 184.511,Z 226.536,A -85,B 0,C 180,E1 -24442.153,E2 -24442.153} C_VEL
LIN {X 0,Y 187.387,Z 214.857,A -85,B 0,C 180,E1 -24443.284,E2 -24443.284} C_VEL
LIN {X 0,Y 189.717,Z 201.923,A -85,B 0,C 180,E1 -24444.141,E2 -24444.141} C_VEL
LIN {X 0,Y 191.089,Z 187.886,A -85,B 0,C 180,E1 -24444.721,E2 -24444.721} C_VEL
LIN {X 0,Y 192.524,Z 167.049,A -85,B 0,C 180,E1 -24445.413,E2 -24445.413} C_VEL
LIN {X 0,Y 187.302,Z 157.025,A -85,B 0,C 180,E1 -24448.152,E2 -24448.152} C_VEL
LIN {X 0,Y 182.086,Z 148.028,A -85,B 0,C 180,E1 -24451.192,E2 -24451.192} C_VEL
LIN {X 0,Y 177.151,Z 140.481,A -85,B 0,C 180,E1 -24454.436,E2 -24454.436} C_VEL
LIN {X 0,Y 174.086,Z 136.125,A -85,B 0,C 180,E1 -24456.706,E2 -24456.706} C_VEL
LIN {X 0,Y 171.404,Z 132.348,A -85,B 0,C 180,E1 -24458.926,E2 -24458.926} C_VEL
LIN {X 0,Y 168.228,Z 127.985,A -85,B 0,C 180,E1 -24461.927,E2 -24461.927} C_VEL
LIN {X 0,Y 165.632,Z 124.73,A -85,B 0,C 180,E1 -24464.778,E2 -24464.778} C_VEL
LIN {X 0,Y 164.728,Z 123.208,A -85,B 0,C 180,E1 -24465.956,E2 -24465.956} C_VEL
LIN {X 0,Y 162.272,Z 120.97,A -85,B 0,C 180,E1 -24469.393,E2 -24469.393} C_VEL
LIN {X 0,Y 160.783,Z 117.751,A -85,B 0,C 180,E1 -24472.464,E2 -24472.464} C_VEL
LIN {X 0,Y 158.414,Z 115.972,A -85,B 0,C 180,E1 -24479.999,E2 -24479.999} C_VEL
LIN {X 0,Y 158.702,Z 116.676,A -85,B 0,C 180,E1 -24488.274,E2 -24488.274} C_VEL
LIN {X 0,Y 160.8,Z 118.083,A -85,B 0,C 180,E1 -24494.07,E2 -24494.07} C_VEL
LIN {X 0,Y 162.153,Z 120.897,A -85,B 0,C 180,E1 -24496.848,E2 -24496.848} C_VEL
LIN {X 0,Y 164.642,Z 123.229,A -85,B 0,C 180,E1 -24500.374,E2 -24500.374} C_VEL
LIN {X 0,Y 167.577,Z 127.425,A -85,B 0,C 180,E1 -24503.857,E2 -24503.857} C_VEL
LIN {X 0,Y 169.423,Z 130.11,A -85,B 0,C 180,E1 -24505.738,E2 -24505.738} C_VEL
LIN {X 0,Y 172.982,Z 136.027,A -85,B 0,C 180,E1 -24508.972,E2 -24508.972} C_VEL
LIN {X 0,Y 175.949,Z 141.233,A -85,B 0,C 180,E1 -24511.336,E2 -24511.336} C_VEL
LIN {X 0,Y 179.392,Z 147.63,A -85,B 0,C 180,E1 -24513.81,E2 -24513.81} C_VEL
LIN {X 0,Y 184.022,Z 156.905,A -85,B 0,C 180,E1 -24516.794,E2 -24516.794} C_VEL
LIN {X 0,Y 188.726,Z 167.84,A -85,B 0,C 180,E1 -24519.563,E2 -24519.563} C_VEL
LIN {X 0,Y 191.911,Z 176.376,A -85,B 0,C 180,E1 -24521.333,E2 -24521.333} C_VEL
LIN {X 0,Y 189.417,Z 208.373,A -85,B 0,C 180,E1 -24522.394,E2 -24522.394} C_VEL
LIN {X 0,Y 187.266,Z 221.856,A -85,B 0,C 180,E1 -24523.139,E2 -24523.139} C_VEL
LIN {X 0,Y 184.276,Z 234.328,A -85,B 0,C 180,E1 -24524.152,E2 -24524.152} C_VEL
LIN {X 0,Y 180.428,Z 246.171,A -85,B 0,C 180,E1 -24525.481,E2 -24525.481} C_VEL
LIN {X 0,Y 175.868,Z 257.561,A -85,B 0,C 180,E1 -24527.206,E2 -24527.206} C_VEL
LIN {X 0,Y 171.123,Z 267.841,A -85,B 0,C 180,E1 -24529.308,E2 -24529.308} C_VEL
LIN {X 0,Y 166.608,Z 276.261,A -85,B 0,C 180,E1 -24531.522,E2 -24531.522} C_VEL
LIN {X 0,Y 161.017,Z 285.41,A -85,B 0,C 180,E1 -24534.666,E2 -24534.666} C_VEL
LIN {X 0,Y 156.004,Z 292.796,A -85,B 0,C 180,E1 -24538.038,E2 -24538.038} C_VEL
LIN {X 0,Y 151.142,Z 299.624,A -85,B 0,C 180,E1 -24542.289,E2 -24542.289} C_VEL
LIN {X 0,Y 147.596,Z 304.153,A -85,B 0,C 180,E1 -24546.124,E2 -24546.124} C_VEL
LIN {X 0,Y 144.722,Z 307.618,A -85,B 0,C 180,E1 -24550.126,E2 -24550.126} C_VEL
LIN {X 0,Y 142.579,Z 310.058,A -85,B 0,C 180,E1 -24554.333,E2 -24554.333} C_VEL
LIN {X 0,Y 141.137,Z 311.079,A -85,B 0,C 180,E1 -24556.614,E2 -24556.614} C_VEL
LIN {X 0,Y 137.403,Z 311.945,A -85,B 0,C 180,E1 -24560.376,E2 -24560.376} C_VEL
LIN {X 0,Y 134.661,Z 312.095,A -85,B 0,C 180,E1 -24563.53,E2 -24563.53} C_VEL
LIN {X 0,Y 133.625,Z 311.903,A -85,B 0,C 180,E1 -24566.028,E2 -24566.028} C_VEL
LIN {X 0,Y 133.594,Z 311.771,A -85,B 0,C 180,E1 -24566.876,E2 -24566.876} C_VEL
LIN {X 0,Y 133.776,Z 311.105,A -85,B 0,C 180,E1 -24569.999,E2 -24569.999} C_VEL
LIN {X 0,Y 133.635,Z 310.009,A -85,B 0,C 180,E1 -24573.014,E2 -24573.014} C_VEL
LIN {X 0,Y 133.582,Z 308.449,A -85,B 0,C 180,E1 -24576.039,E2 -24576.039} C_VEL
LIN {X 0,Y 134.017,Z 305.309,A -85,B 0,C 180,E1 -24580.575,E2 -24580.575} C_VEL
LIN {X 0,Y 134.995,Z 301.081,A -85,B 0,C 180,E1 -24585.087,E2 -24585.087} C_VEL
LIN {X 0,Y 137.285,Z 294.654,A -85,B 0,C 180,E1 -24590.215,E2 -24590.215} C_VEL
LIN {X 0,Y 140.001,Z 287.77,A -85,B 0,C 180,E1 -24594.387,E2 -24594.387} C_VEL
LIN {X 0,Y 142.516,Z 280.758,A -85,B 0,C 180,E1 -24597.775,E2 -24597.775} C_VEL
LIN {X 0,Y 145.853,Z 271.75,A -85,B 0,C 180,E1 -24601.197,E2 -24601.197} C_VEL
LIN {X 0,Y 149.33,Z 262.237,A -85,B 0,C 180,E1 -24603.977,E2 -24603.977} C_VEL
LIN {X 0,Y 152.673,Z 251.858,A -85,B 0,C 180,E1 -24606.346,E2 -24606.346} C_VEL
LIN {X 0,Y 155.825,Z 240.485,A -85,B 0,C 180,E1 -24608.326,E2 -24608.326} C_VEL
LIN {X 0,Y 158.5,Z 228.886,A -85,B 0,C 180,E1 -24609.803,E2 -24609.803} C_VEL
LIN {X 0,Y 160.593,Z 215.456,A -85,B 0,C 180,E1 -24611.028,E2 -24611.028} C_VEL
LIN {X 0,Y 161.935,Z 201.793,A -85,B 0,C 180,E1 -24611.785,E2 -24611.785} C_VEL
LIN {X 0,Y 164.015,Z 166.044,A -85,B 0,C 180,E1 -24613.182,E2 -24613.182} C_VEL
LIN {X 0,Y 162.862,Z 151.275,A -85,B 0,C 180,E1 -24614.356,E2 -24614.356} C_VEL
LIN {X 0,Y 158.392,Z 139.189,A -85,B 0,C 180,E1 -24616.494,E2 -24616.494} C_VEL
LIN {X 0,Y 153.033,Z 127.389,A -85,B 0,C 180,E1 -24619.156,E2 -24619.156} C_VEL
LIN {X 0,Y 147.634,Z 117.306,A -85,B 0,C 180,E1 -24622.054,E2 -24622.054} C_VEL
LIN {X 0,Y 145.783,Z 114.473,A -85,B 0,C 180,E1 -24623.09,E2 -24623.09} C_VEL
LIN {X 0,Y 142.733,Z 110.309,A -85,B 0,C 180,E1 -24624.868,E2 -24624.868} C_VEL
LIN {X 0,Y 140.408,Z 107.285,A -85,B 0,C 180,E1 -24626.311,E2 -24626.311} C_VEL
LIN {X 0,Y 139.543,Z 105.751,A -85,B 0,C 180,E1 -24626.908,E2 -24626.908} C_VEL
LIN {X 0,Y 137.192,Z 103.578,A -85,B 0,C 180,E1 -24628.435,E2 -24628.435} C_VEL
LIN {X 0,Y 136.158,Z 101.192,A -85,B 0,C 180,E1 -24629.272,E2 -24629.272} C_VEL
LIN {X 0,Y 136.052,Z 100.536,A -85,B 0,C 180,E1 -24629.419,E2 -24629.419} C_VEL
LIN {X 0,Y 136.145,Z 100.513,A -85,B 0,C 180,E1 -24632.317,E2 -24632.317} C_VEL
LIN {X 0,Y 136.243,Z 100.495,A -85,B 0,C 180,E1 -24638.833,E2 -24638.833} C_VEL
LIN {X 0,Y 136.268,Z 100.501,A -85,B 0,C 180,E1 -24645.057,E2 -24645.057} C_VEL
LIN {X 0,Y 136.444,Z 100.463,A -85,B 0,C 180,E1 -24648.138,E2 -24648.138} C_VEL
LIN {X 0,Y 136.551,Z 100.474,A -85,B 0,C 180,E1 -24651.118,E2 -24651.118} C_VEL
LIN {X 0,Y 137.13,Z 100.402,A -85,B 0,C 180,E1 -24660.001,E2 -24660.001} C_VEL
LIN {X 0,Y 136.548,Z 100.473,A -85,B 0,C 180,E1 -24668.883,E2 -24668.883} C_VEL
LIN {X 0,Y 136.417,Z 100.468,A -85,B 0,C 180,E1 -24671.893,E2 -24671.893} C_VEL
LIN {X 0,Y 136.238,Z 100.51,A -85,B 0,C 180,E1 -24678.031,E2 -24678.031} C_VEL
LIN {X 0,Y 136.198,Z 100.494,A -85,B 0,C 180,E1 -24681.75,E2 -24681.75} C_VEL
LIN {X 0,Y 136.1,Z 100.53,A -85,B 0,C 180,E1 -24688.617,E2 -24688.617} C_VEL
LIN {X 0,Y 136.042,Z 100.535,A -85,B 0,C 180,E1 -24694.631,E2 -24694.631} C_VEL
LIN {X 0,Y 136.047,Z 100.727,A -85,B 0,C 180,E1 -24698.31,E2 -24698.31} C_VEL
LIN {X 0,Y 136.974,Z 103.339,A -85,B 0,C 180,E1 -24699.11,E2 -24699.11} C_VEL
LIN {X 0,Y 139.032,Z 105.495,A -85,B 0,C 180,E1 -24700.483,E2 -24700.483} C_VEL
LIN {X 0,Y 139.916,Z 106.365,A -85,B 0,C 180,E1 -24701.043,E2 -24701.043} C_VEL
LIN {X 0,Y 141.849,Z 109.479,A -85,B 0,C 180,E1 -24702.317,E2 -24702.317} C_VEL
LIN {X 0,Y 143.573,Z 111.431,A -85,B 0,C 180,E1 -24703.333,E2 -24703.333} C_VEL
LIN {X 0,Y 147.26,Z 116.796,A -85,B 0,C 180,E1 -24705.444,E2 -24705.444} C_VEL
LIN {X 0,Y 151.41,Z 122.831,A -85,B 0,C 180,E1 -24707.605,E2 -24707.605} C_VEL
LIN {X 0,Y 157.892,Z 133.722,A -85,B 0,C 180,E1 -24710.701,E2 -24710.701} C_VEL
LIN {X 0,Y 164.208,Z 146.415,A -85,B 0,C 180,E1 -24713.472,E2 -24713.472} C_VEL
LIN {X 0,Y 165.003,Z 148.267,A -85,B 0,C 180,E1 -24713.812,E2 -24713.812} C_VEL
LIN {X 0,Y 161.966,Z 197.314,A -85,B 0,C 180,E1 -24715.779,E2 -24715.779} C_VEL
LIN {X 0,Y 160.313,Z 211.142,A -85,B 0,C 180,E1 -24716.826,E2 -24716.826} C_VEL
LIN {X 0,Y 158.304,Z 222.991,A -85,B 0,C 180,E1 -24718.184,E2 -24718.184} C_VEL
LIN {X 0,Y 155.442,Z 235.571,A -85,B 0,C 180,E1 -24720.177,E2 -24720.177} C_VEL
LIN {X 0,Y 152.272,Z 246.764,A -85,B 0,C 180,E1 -24722.514,E2 -24722.514} C_VEL
LIN {X 0,Y 148.911,Z 256.863,A -85,B 0,C 180,E1 -24725.238,E2 -24725.238} C_VEL
LIN {X 0,Y 145.155,Z 266.772,A -85,B 0,C 180,E1 -24728.708,E2 -24728.708} C_VEL
LIN {X 0,Y 141.727,Z 275.489,A -85,B 0,C 180,E1 -24732.692,E2 -24732.692} C_VEL
LIN {X 0,Y 138.909,Z 282.459,A -85,B 0,C 180,E1 -24736.841,E2 -24736.841} C_VEL
LIN {X 0,Y 136.677,Z 288.037,A -85,B 0,C 180,E1 -24741.127,E2 -24741.127} C_VEL
LIN {X 0,Y 135.092,Z 292.431,A -85,B 0,C 180,E1 -24745.525,E2 -24745.525} C_VEL
LIN {X 0,Y 134.2,Z 295.762,A -85,B 0,C 180,E1 -24750.001,E2 -24750.001} C_VEL
LIN {X 0,Y 133.89,Z 297.982,A -85,B 0,C 180,E1 -24754.176,E2 -24754.176} C_VEL
LIN {X 0,Y 133.706,Z 299.578,A -85,B 0,C 180,E1 -24759.074,E2 -24759.074} C_VEL
LIN {X 0,Y 133.966,Z 300.025,A -85,B 0,C 180,E1 -24762.114,E2 -24762.114} C_VEL
LIN {X 0,Y 135.373,Z 299.756,A -85,B 0,C 180,E1 -24768.15,E2 -24768.15} C_VEL
LIN {X 0,Y 137.587,Z 298.27,A -85,B 0,C 180,E1 -24773.153,E2 -24773.153} C_VEL
LIN {X 0,Y 139.765,Z 296.286,A -85,B 0,C 180,E1 -24776.909,E2 -24776.909} C_VEL
LIN {X 0,Y 142.955,Z 293.089,A -85,B 0,C 180,E1 -24781.079,E2 -24781.079} C_VEL
LIN {X 0,Y 146.774,Z 288.802,A -85,B 0,C 180,E1 -24785.072,E2 -24785.072} C_VEL
LIN {X 0,Y 151.318,Z 283.296,A -85,B 0,C 180,E1 -24788.831,E2 -24788.831} C_VEL
LIN {X 0,Y 156.418,Z 276.388,A -85,B 0,C 180,E1 -24792.375,E2 -24792.375} C_VEL
LIN {X 0,Y 161.559,Z 268.415,A -85,B 0,C 180,E1 -24795.472,E2 -24795.472} C_VEL
LIN {X 0,Y 166.913,Z 258.713,A -85,B 0,C 180,E1 -24798.365,E2 -24798.365} C_VEL
LIN {X 0,Y 171.764,Z 248.825,A -85,B 0,C 180,E1 -24800.562,E2 -24800.562} C_VEL
LIN {X 0,Y 176.276,Z 237.856,A -85,B 0,C 180,E1 -24802.412,E2 -24802.412} C_VEL
LIN {X 0,Y 180.191,Z 225.8,A -85,B 0,C 180,E1 -24803.956,E2 -24803.956} C_VEL
LIN {X 0,Y 182.678,Z 215.999,A -85,B 0,C 180,E1 -24804.906,E2 -24804.906} C_VEL
LIN {X 0,Y 185.12,Z 203.258,A -85,B 0,C 180,E1 -24805.769,E2 -24805.769} C_VEL
LIN {X 0,Y 186.528,Z 190.558,A -85,B 0,C 180,E1 -24806.335,E2 -24806.335} C_VEL
LIN {X 0,Y 188.073,Z 170.054,A -85,B 0,C 180,E1 -24806.991,E2 -24806.991} C_VEL
LIN {X 0,Y 182.434,Z 159.232,A -85,B 0,C 180,E1 -24810.219,E2 -24810.219} C_VEL
LIN {X 0,Y 177.329,Z 150.531,A -85,B 0,C 180,E1 -24813.521,E2 -24813.521} C_VEL
LIN {X 0,Y 172.412,Z 142.958,A -85,B 0,C 180,E1 -24817.196,E2 -24817.196} C_VEL
LIN {X 0,Y 169.265,Z 138.514,A -85,B 0,C 180,E1 -24819.918,E2 -24819.918} C_VEL
LIN {X 0,Y 166.399,Z 134.417,A -85,B 0,C 180,E1 -24822.803,E2 -24822.803} C_VEL
LIN {X 0,Y 163.882,Z 130.974,A -85,B 0,C 180,E1 -24825.783,E2 -24825.783} C_VEL
LIN {X 0,Y 163.271,Z 129.993,A -85,B 0,C 180,E1 -24826.622,E2 -24826.622} C_VEL
LIN {X 0,Y 160.824,Z 127.45,A -85,B 0,C 180,E1 -24830.329,E2 -24830.329} C_VEL
LIN {X 0,Y 159.615,Z 124.679,A -85,B 0,C 180,E1 -24833.045,E2 -24833.045} C_VEL
LIN {X 0,Y 157.545,Z 123.028,A -85,B 0,C 180,E1 -24839.999,E2 -24839.999} C_VEL
LIN {X 0,Y 157.84,Z 123.741,A -85,B 0,C 180,E1 -24848.32,E2 -24848.32} C_VEL
LIN {X 0,Y 159.645,Z 125.021,A -85,B 0,C 180,E1 -24853.525,E2 -24853.525} C_VEL
LIN {X 0,Y 161.025,Z 127.834,A -85,B 0,C 180,E1 -24856.479,E2 -24856.479} C_VEL
LIN {X 0,Y 163.558,Z 130.495,A -85,B 0,C 180,E1 -24860.208,E2 -24860.208} C_VEL
LIN {X 0,Y 165.855,Z 133.933,A -85,B 0,C 180,E1 -24863.054,E2 -24863.054} C_VEL
LIN {X 0,Y 167.481,Z 136.365,A -85,B 0,C 180,E1 -24864.811,E2 -24864.811} C_VEL
LIN {X 0,Y 170.808,Z 142.183,A -85,B 0,C 180,E1 -24868.035,E2 -24868.035} C_VEL
LIN {X 0,Y 173.744,Z 147.6,A -85,B 0,C 180,E1 -24870.521,E2 -24870.521} C_VEL
LIN {X 0,Y 177.508,Z 154.987,A -85,B 0,C 180,E1 -24873.356,E2 -24873.356} C_VEL
LIN {X 0,Y 181.474,Z 163.586,A -85,B 0,C 180,E1 -24876.051,E2 -24876.051} C_VEL
LIN {X 0,Y 185.344,Z 173,A -85,B 0,C 180,E1 -24878.47,E2 -24878.47} C_VEL
LIN {X 0,Y 187.394,Z 178.801,A -85,B 0,C 180,E1 -24879.706,E2 -24879.706} C_VEL
LIN {X 0,Y 184.972,Z 208.414,A -85,B 0,C 180,E1 -24880.704,E2 -24880.704} C_VEL
LIN {X 0,Y 182.834,Z 221.342,A -85,B 0,C 180,E1 -24881.417,E2 -24881.417} C_VEL
LIN {X 0,Y 179.723,Z 233.93,A -85,B 0,C 180,E1 -24882.429,E2 -24882.429} C_VEL
LIN {X 0,Y 175.454,Z 246.58,A -85,B 0,C 180,E1 -24883.861,E2 -24883.861} C_VEL
LIN {X 0,Y 170.73,Z 257.837,A -85,B 0,C 180,E1 -24885.589,E2 -24885.589} C_VEL
LIN {X 0,Y 165.788,Z 267.991,A -85,B 0,C 180,E1 -24887.703,E2 -24887.703} C_VEL
LIN {X 0,Y 160.093,Z 277.96,A -85,B 0,C 180,E1 -24890.464,E2 -24890.464} C_VEL
LIN {X 0,Y 154.358,Z 286.759,A -85,B 0,C 180,E1 -24893.707,E2 -24893.707} C_VEL
LIN {X 0,Y 149.219,Z 293.82,A -85,B 0,C 180,E1 -24897.204,E2 -24897.204} C_VEL
LIN {X 0,Y 144.871,Z 299.489,A -85,B 0,C 180,E1 -24900.979,E2 -24900.979} C_VEL
LIN {X 0,Y 141.117,Z 303.974,A -85,B 0,C 180,E1 -24904.954,E2 -24904.954} C_VEL
LIN {X 0,Y 138.044,Z 307.4,A -85,B 0,C 180,E1 -24909.121,E2 -24909.121} C_VEL
LIN {X 0,Y 135.577,Z 309.974,A -85,B 0,C 180,E1 -24913.887,E2 -24913.887} C_VEL
LIN {X 0,Y 134.331,Z 311.382,A -85,B 0,C 180,E1 -24917.919,E2 -24917.919} C_VEL
LIN {X 0,Y 133.797,Z 311.909,A -85,B 0,C 180,E1 -24920.932,E2 -24920.932} C_VEL
LIN {X 0,Y 133.594,Z 311.771,A -85,B 0,C 180,E1 -24926.876,E2 -24926.876} C_VEL
LIN {X 0,Y 133.362,Z 311.518,A -85,B 0,C 180,E1 -24928.552,E2 -24928.552} C_VEL
LIN {X 0,Y 132.034,Z 310.804,A -85,B 0,C 180,E1 -24931.022,E2 -24931.022} C_VEL
LIN {X 0,Y 128.82,Z 308.881,A -85,B 0,C 180,E1 -24935.108,E2 -24935.108} C_VEL
LIN {X 0,Y 126.982,Z 306.762,A -85,B 0,C 180,E1 -24938.505,E2 -24938.505} C_VEL
LIN {X 0,Y 126.851,Z 305.535,A -85,B 0,C 180,E1 -24940.234,E2 -24940.234} C_VEL
LIN {X 0,Y 127.653,Z 302.125,A -85,B 0,C 180,E1 -24944.343,E2 -24944.343} C_VEL
LIN {X 0,Y 129.393,Z 297.087,A -85,B 0,C 180,E1 -24949.019,E2 -24949.019} C_VEL
LIN {X 0,Y 131.909,Z 290.75,A -85,B 0,C 180,E1 -24953.552,E2 -24953.552} C_VEL
LIN {X 0,Y 134.285,Z 284.751,A -85,B 0,C 180,E1 -24956.948,E2 -24956.948} C_VEL
LIN {X 0,Y 137.612,Z 276.455,A -85,B 0,C 180,E1 -24960.71,E2 -24960.71} C_VEL
LIN {X 0,Y 141.318,Z 266.943,A -85,B 0,C 180,E1 -24964.019,E2 -24964.019} C_VEL
LIN {X 0,Y 145.257,Z 256.41,A -85,B 0,C 180,E1 -24966.779,E2 -24966.779} C_VEL
LIN {X 0,Y 148.405,Z 246.254,A -85,B 0,C 180,E1 -24968.863,E2 -24968.863} C_VEL
LIN {X 0,Y 151.578,Z 234.34,A -85,B 0,C 180,E1 -24970.693,E2 -24970.693} C_VEL
LIN {X 0,Y 154.052,Z 221.875,A -85,B 0,C 180,E1 -24972.07,E2 -24972.07} C_VEL
LIN {X 0,Y 155.9,Z 208.396,A -85,B 0,C 180,E1 -24973.054,E2 -24973.054} C_VEL
LIN {X 0,Y 158.569,Z 166.896,A -85,B 0,C 180,E1 -24974.777,E2 -24974.777} C_VEL
LIN {X 0,Y 157.637,Z 153.797,A -85,B 0,C 180,E1 -24975.861,E2 -24975.861} C_VEL
LIN {X 0,Y 153.772,Z 143.103,A -85,B 0,C 180,E1 -24977.863,E2 -24977.863} C_VEL
LIN {X 0,Y 148.861,Z 131.949,A -85,B 0,C 180,E1 -24980.501,E2 -24980.501} C_VEL
LIN {X 0,Y 143.871,Z 122.287,A -85,B 0,C 180,E1 -24983.392,E2 -24983.392} C_VEL
LIN {X 0,Y 141.663,Z 119.052,A -85,B 0,C 180,E1 -24984.712,E2 -24984.712} C_VEL
LIN {X 0,Y 139.366,Z 115.834,A -85,B 0,C 180,E1 -24986.16,E2 -24986.16} C_VEL
LIN {X 0,Y 136.899,Z 112.212,A -85,B 0,C 180,E1 -24987.842,E2 -24987.842} C_VEL
LIN {X 0,Y 133.905,Z 108.732,A -85,B 0,C 180,E1 -24989.984,E2 -24989.984} C_VEL
LIN {X 0,Y 132.851,Z 106.85,A -85,B 0,C 180,E1 -24990.855,E2 -24990.855} C_VEL
LIN {X 0,Y 130.445,Z 104.795,A -85,B 0,C 180,E1 -24992.745,E2 -24992.745} C_VEL
LIN {X 0,Y 129.171,Z 102.238,A -85,B 0,C 180,E1 -24993.982,E2 -24993.982} C_VEL
LIN {X 0,Y 129.021,Z 101.4,A -85,B 0,C 180,E1 -24994.274,E2 -24994.274} C_VEL
LIN {X 0,Y 129.106,Z 101.392,A -85,B 0,C 180,E1 -24997.728,E2 -24997.728} C_VEL
LIN {X 0,Y 129.152,Z 101.378,A -85,B 0,C 180,E1 -25000.944,E2 -25000.944} C_VEL
LIN {X 0,Y 129.365,Z 101.343,A -85,B 0,C 180,E1 -25007.924,E2 -25007.924} C_VEL
LIN {X 0,Y 129.476,Z 101.351,A -85,B 0,C 180,E1 -25010.629,E2 -25010.629} C_VEL
LIN {X 0,Y 130.085,Z 101.279,A -85,B 0,C 180,E1 -25020.001,E2 -25020.001} C_VEL
LIN {X 0,Y 129.471,Z 101.354,A -85,B 0,C 180,E1 -25029.373,E2 -25029.373} C_VEL
LIN {X 0,Y 129.179,Z 101.381,A -85,B 0,C 180,E1 -25035.786,E2 -25035.786} C_VEL
LIN {X 0,Y 129.151,Z 101.383,A -85,B 0,C 180,E1 -25039.057,E2 -25039.057} C_VEL
LIN {X 0,Y 129.108,Z 101.378,A -85,B 0,C 180,E1 -25042.399,E2 -25042.399} C_VEL
LIN {X 0,Y 129.036,Z 101.412,A -85,B 0,C 180,E1 -25049.374,E2 -25049.374} C_VEL
LIN {X 0,Y 128.994,Z 101.423,A -85,B 0,C 180,E1 -25053.486,E2 -25053.486} C_VEL
LIN {X 0,Y 129.754,Z 103.768,A -85,B 0,C 180,E1 -25054.327,E2 -25054.327} C_VEL
LIN {X 0,Y 131.313,Z 105.847,A -85,B 0,C 180,E1 -25055.682,E2 -25055.682} C_VEL
LIN {X 0,Y 133.103,Z 107.123,A -85,B 0,C 180,E1 -25057.033,E2 -25057.033} C_VEL
LIN {X 0,Y 134.881,Z 110.212,A -85,B 0,C 180,E1 -25058.464,E2 -25058.464} C_VEL
LIN {X 0,Y 136.828,Z 112.218,A -85,B 0,C 180,E1 -25059.812,E2 -25059.812} C_VEL
LIN {X 0,Y 139.343,Z 115.853,A -85,B 0,C 180,E1 -25061.526,E2 -25061.526} C_VEL
LIN {X 0,Y 143.429,Z 121.625,A -85,B 0,C 180,E1 -25064.048,E2 -25064.048} C_VEL
LIN {X 0,Y 148.1,Z 128.821,A -85,B 0,C 180,E1 -25066.664,E2 -25066.664} C_VEL
LIN {X 0,Y 153.608,Z 138.256,A -85,B 0,C 180,E1 -25069.465,E2 -25069.465} C_VEL
LIN {X 0,Y 159.558,Z 150.602,A -85,B 0,C 180,E1 -25072.273,E2 -25072.273} C_VEL
LIN {X 0,Y 156.51,Z 197.065,A -85,B 0,C 180,E1 -25074.15,E2 -25074.15} C_VEL
LIN {X 0,Y 154.845,Z 210.441,A -85,B 0,C 180,E1 -25075.149,E2 -25075.149} C_VEL
LIN {X 0,Y 152.591,Z 223.373,A -85,B 0,C 180,E1 -25076.647,E2 -25076.647} C_VEL
LIN {X 0,Y 149.785,Z 235.154,A -85,B 0,C 180,E1 -25078.535,E2 -25078.535} C_VEL
LIN {X 0,Y 146.453,Z 246.48,A -85,B 0,C 180,E1 -25080.931,E2 -25080.931} C_VEL
LIN {X 0,Y 142.914,Z 256.707,A -85,B 0,C 180,E1 -25083.732,E2 -25083.732} C_VEL
LIN {X 0,Y 139.283,Z 265.9,A -85,B 0,C 180,E1 -25086.981,E2 -25086.981} C_VEL
LIN {X 0,Y 135.561,Z 274.818,A -85,B 0,C 180,E1 -25091.095,E2 -25091.095} C_VEL
LIN {X 0,Y 132.496,Z 282.004,A -85,B 0,C 180,E1 -25095.408,E2 -25095.408} C_VEL
LIN {X 0,Y 130.397,Z 286.864,A -85,B 0,C 180,E1 -25099.128,E2 -25099.128} C_VEL
LIN {X 0,Y 128.495,Z 291.591,A -85,B 0,C 180,E1 -25103.721,E2 -25103.721} C_VEL
LIN {X 0,Y 127.39,Z 295.212,A -85,B 0,C 180,E1 -25108.42,E2 -25108.42} C_VEL
LIN {X 0,Y 126.799,Z 298.167,A -85,B 0,C 180,E1 -25113.893,E2 -25113.893} C_VEL
LIN {X 0,Y 126.629,Z 299.939,A -85,B 0,C 180,E1 -25119.586,E2 -25119.586} C_VEL
LIN {X 0,Y 127.546,Z 300.399,A -85,B 0,C 180,E1 -25125.993,E2 -25125.993} C_VEL
LIN {X 0,Y 128.577,Z 300.048,A -85,B 0,C 180,E1 -25129.146,E2 -25129.146} C_VEL
LIN {X 0,Y 130.806,Z 298.652,A -85,B 0,C 180,E1 -25134.021,E2 -25134.021} C_VEL
LIN {X 0,Y 134.451,Z 295.527,A -85,B 0,C 180,E1 -25139.775,E2 -25139.775} C_VEL
LIN {X 0,Y 138.135,Z 291.932,A -85,B 0,C 180,E1 -25144.033,E2 -25144.033} C_VEL
LIN {X 0,Y 142.68,Z 286.975,A -85,B 0,C 180,E1 -25148.225,E2 -25148.225} C_VEL
LIN {X 0,Y 148.412,Z 280.057,A -85,B 0,C 180,E1 -25152.44,E2 -25152.44} C_VEL
LIN {X 0,Y 154.077,Z 272.213,A -85,B 0,C 180,E1 -25155.925,E2 -25155.925} C_VEL
LIN {X 0,Y 159.054,Z 264.165,A -85,B 0,C 180,E1 -25158.693,E2 -25158.693} C_VEL
LIN {X 0,Y 164.437,Z 254.31,A -85,B 0,C 180,E1 -25161.262,E2 -25161.262} C_VEL
LIN {X 0,Y 169.629,Z 243.253,A -85,B 0,C 180,E1 -25163.394,E2 -25163.394} C_VEL
LIN {X 0,Y 174.024,Z 231.658,A -85,B 0,C 180,E1 -25165.065,E2 -25165.065} C_VEL
LIN {X 0,Y 177.318,Z 220.286,A -85,B 0,C 180,E1 -25166.341,E2 -25166.341} C_VEL
LIN {X 0,Y 180.187,Z 207.474,A -85,B 0,C 180,E1 -25167.319,E2 -25167.319} C_VEL
LIN {X 0,Y 181.974,Z 194.618,A -85,B 0,C 180,E1 -25167.96,E2 -25167.96} C_VEL
LIN {X 0,Y 183.664,Z 172.979,A -85,B 0,C 180,E1 -25168.7,E2 -25168.7} C_VEL
LIN {X 0,Y 178.249,Z 162.45,A -85,B 0,C 180,E1 -25172.091,E2 -25172.091} C_VEL
LIN {X 0,Y 173.634,Z 154.603,A -85,B 0,C 180,E1 -25175.362,E2 -25175.362} C_VEL
LIN {X 0,Y 169.737,Z 148.456,A -85,B 0,C 180,E1 -25178.55,E2 -25178.55} C_VEL
LIN {X 0,Y 167.335,Z 144.871,A -85,B 0,C 180,E1 -25180.785,E2 -25180.785} C_VEL
LIN {X 0,Y 164.683,Z 140.937,A -85,B 0,C 180,E1 -25183.616,E2 -25183.616} C_VEL
LIN {X 0,Y 162.159,Z 137.171,A -85,B 0,C 180,E1 -25186.847,E2 -25186.847} C_VEL
LIN {X 0,Y 159.394,Z 133.85,A -85,B 0,C 180,E1 -25191.342,E2 -25191.342} C_VEL
LIN {X 0,Y 158.463,Z 131.613,A -85,B 0,C 180,E1 -25193.634,E2 -25193.634} C_VEL
LIN {X 0,Y 156.672,Z 130.104,A -85,B 0,C 180,E1 -25199.999,E2 -25199.999} C_VEL
LIN {X 0,Y 156.848,Z 130.655,A -85,B 0,C 180,E1 -25207.725,E2 -25207.725} C_VEL
LIN {X 0,Y 158.523,Z 131.968,A -85,B 0,C 180,E1 -25213.01,E2 -25213.01} C_VEL
LIN {X 0,Y 159.936,Z 134.815,A -85,B 0,C 180,E1 -25216.162,E2 -25216.162} C_VEL
LIN {X 0,Y 162.156,Z 137.335,A -85,B 0,C 180,E1 -25219.599,E2 -25219.599} C_VEL
LIN {X 0,Y 165.521,Z 142.549,A -85,B 0,C 180,E1 -25223.797,E2 -25223.797} C_VEL
LIN {X 0,Y 168.491,Z 147.972,A -85,B 0,C 180,E1 -25226.891,E2 -25226.891} C_VEL
LIN {X 0,Y 171.701,Z 154.241,A -85,B 0,C 180,E1 -25229.792,E2 -25229.792} C_VEL
LIN {X 0,Y 175.976,Z 163.194,A -85,B 0,C 180,E1 -25233.155,E2 -25233.155} C_VEL
LIN {X 0,Y 180.317,Z 173.668,A -85,B 0,C 180,E1 -25236.208,E2 -25236.208} C_VEL
LIN {X 0,Y 183.03,Z 181.243,A -85,B 0,C 180,E1 -25237.997,E2 -25237.997} C_VEL
LIN {X 0,Y 180.832,Z 207.437,A -85,B 0,C 180,E1 -25238.886,E2 -25238.886} C_VEL
LIN {X 0,Y 178.572,Z 220.776,A -85,B 0,C 180,E1 -25239.601,E2 -25239.601} C_VEL
LIN {X 0,Y 175.349,Z 233.531,A -85,B 0,C 180,E1 -25240.621,E2 -25240.621} C_VEL
LIN {X 0,Y 171.254,Z 245.41,A -85,B 0,C 180,E1 -25241.941,E2 -25241.941} C_VEL
LIN {X 0,Y 166.363,Z 256.822,A -85,B 0,C 180,E1 -25243.659,E2 -25243.659} C_VEL
LIN {X 0,Y 161.154,Z 267.121,A -85,B 0,C 180,E1 -25245.751,E2 -25245.751} C_VEL
LIN {X 0,Y 155.755,Z 276.386,A -85,B 0,C 180,E1 -25248.274,E2 -25248.274} C_VEL
LIN {X 0,Y 149.623,Z 285.393,A -85,B 0,C 180,E1 -25251.51,E2 -25251.51} C_VEL
LIN {X 0,Y 144.125,Z 292.669,A -85,B 0,C 180,E1 -25255.041,E2 -25255.041} C_VEL
LIN {X 0,Y 138.691,Z 299.353,A -85,B 0,C 180,E1 -25259.552,E2 -25259.552} C_VEL
LIN {X 0,Y 134.706,Z 303.796,A -85,B 0,C 180,E1 -25263.674,E2 -25263.674} C_VEL
LIN {X 0,Y 131.417,Z 307.181,A -85,B 0,C 180,E1 -25268.015,E2 -25268.015} C_VEL
LIN {X 0,Y 129.618,Z 308.879,A -85,B 0,C 180,E1 -25271.014,E2 -25271.014} C_VEL
LIN {X 0,Y 127.369,Z 311.104,A -85,B 0,C 180,E1 -25277.248,E2 -25277.248} C_VEL
LIN {X 0,Y 126.762,Z 311.596,A -85,B 0,C 180,E1 -25280.425,E2 -25280.425} C_VEL
LIN {X 0,Y 126.507,Z 311.397,A -85,B 0,C 180,E1 -25286.91,E2 -25286.91} C_VEL
LIN {X 0,Y 126.681,Z 310.739,A -85,B 0,C 180,E1 -25289.999,E2 -25289.999} C_VEL
LIN {X 0,Y 126.546,Z 309.606,A -85,B 0,C 180,E1 -25293.183,E2 -25293.183} C_VEL
LIN {X 0,Y 126.59,Z 307.102,A -85,B 0,C 180,E1 -25297.977,E2 -25297.977} C_VEL
LIN {X 0,Y 126.851,Z 305.535,A -85,B 0,C 180,E1 -25300.234,E2 -25300.234} C_VEL
LIN {X 0,Y 126.654,Z 303.591,A -85,B 0,C 180,E1 -25302.746,E2 -25302.746} C_VEL
LIN {X 0,Y 125.023,Z 299.829,A -85,B 0,C 180,E1 -25306.86,E2 -25306.86} C_VEL
LIN {X 0,Y 123.849,Z 295.458,A -85,B 0,C 180,E1 -25310.935,E2 -25310.935} C_VEL
LIN {X 0,Y 124.362,Z 292.452,A -85,B 0,C 180,E1 -25313.283,E2 -25313.283} C_VEL
LIN {X 0,Y 127.104,Z 286.321,A -85,B 0,C 180,E1 -25317.17,E2 -25317.17} C_VEL
LIN {X 0,Y 130.792,Z 277.4,A -85,B 0,C 180,E1 -25321.594,E2 -25321.594} C_VEL
LIN {X 0,Y 134.68,Z 268.23,A -85,B 0,C 180,E1 -25325.03,E2 -25325.03} C_VEL
LIN {X 0,Y 138.676,Z 258.088,A -85,B 0,C 180,E1 -25327.914,E2 -25327.914} C_VEL
LIN {X 0,Y 142.418,Z 246.787,A -85,B 0,C 180,E1 -25330.367,E2 -25330.367} C_VEL
LIN {X 0,Y 145.983,Z 234.095,A -85,B 0,C 180,E1 -25332.375,E2 -25332.375} C_VEL
LIN {X 0,Y 148.558,Z 221.663,A -85,B 0,C 180,E1 -25333.778,E2 -25333.778} C_VEL
LIN {X 0,Y 150.486,Z 208.038,A -85,B 0,C 180,E1 -25334.794,E2 -25334.794} C_VEL
LIN {X 0,Y 153.277,Z 168.089,A -85,B 0,C 180,E1 -25336.456,E2 -25336.456} C_VEL
LIN {X 0,Y 152.494,Z 156.235,A -85,B 0,C 180,E1 -25337.484,E2 -25337.484} C_VEL
LIN {X 0,Y 148.636,Z 145.356,A -85,B 0,C 180,E1 -25339.67,E2 -25339.67} C_VEL
LIN {X 0,Y 143.974,Z 134.861,A -85,B 0,C 180,E1 -25342.401,E2 -25342.401} C_VEL
LIN {X 0,Y 140.013,Z 126.953,A -85,B 0,C 180,E1 -25344.915,E2 -25344.915} C_VEL
LIN {X 0,Y 136.343,Z 121.618,A -85,B 0,C 180,E1 -25347.339,E2 -25347.339} C_VEL
LIN {X 0,Y 133.268,Z 117.308,A -85,B 0,C 180,E1 -25349.58,E2 -25349.58} C_VEL
LIN {X 0,Y 130.751,Z 113.918,A -85,B 0,C 180,E1 -25351.586,E2 -25351.586} C_VEL
LIN {X 0,Y 129.92,Z 112.844,A -85,B 0,C 180,E1 -25352.286,E2 -25352.286} C_VEL
LIN {X 0,Y 127.345,Z 109.917,A -85,B 0,C 180,E1 -25354.569,E2 -25354.569} C_VEL
LIN {X 0,Y 126.4,Z 107.991,A -85,B 0,C 180,E1 -25355.573,E2 -25355.573} C_VEL
LIN {X 0,Y 123.724,Z 106.042,A -85,B 0,C 180,E1 -25358.239,E2 -25358.239} C_VEL
LIN {X 0,Y 122.362,Z 103.615,A -85,B 0,C 180,E1 -25359.952,E2 -25359.952} C_VEL
LIN {X 0,Y 122.083,Z 102.256,A -85,B 0,C 180,E1 -25360.561,E2 -25360.561} C_VEL
LIN {X 0,Y 122.316,Z 102.22,A -85,B 0,C 180,E1 -25367.624,E2 -25367.624} C_VEL
LIN {X 0,Y 122.423,Z 102.227,A -85,B 0,C 180,E1 -25373.408,E2 -25373.408} C_VEL
LIN {X 0,Y 123.038,Z 102.157,A -85,B 0,C 180,E1 -25380.001,E2 -25380.001} C_VEL
LIN {X 0,Y 122.404,Z 102.216,A -85,B 0,C 180,E1 -25386.806,E2 -25386.806} C_VEL
LIN {X 0,Y 122.289,Z 102.224,A -85,B 0,C 180,E1 -25392.317,E2 -25392.317} C_VEL
LIN {X 0,Y 122.099,Z 102.271,A -85,B 0,C 180,E1 -25396.727,E2 -25396.727} C_VEL
LIN {X 0,Y 122.023,Z 102.262,A -85,B 0,C 180,E1 -25402.852,E2 -25402.852} C_VEL
LIN {X 0,Y 121.952,Z 102.302,A -85,B 0,C 180,E1 -25407.106,E2 -25407.106} C_VEL
LIN {X 0,Y 122.598,Z 104.528,A -85,B 0,C 180,E1 -25408.117,E2 -25408.117} C_VEL
LIN {X 0,Y 124.857,Z 107.213,A -85,B 0,C 180,E1 -25410.672,E2 -25410.672} C_VEL
LIN {X 0,Y 126.483,Z 108.167,A -85,B 0,C 180,E1 -25412.214,E2 -25412.214} C_VEL
LIN {X 0,Y 128.303,Z 111.393,A -85,B 0,C 180,E1 -25414.049,E2 -25414.049} C_VEL
LIN {X 0,Y 130.566,Z 113.659,A -85,B 0,C 180,E1 -25415.954,E2 -25415.954} C_VEL
LIN {X 0,Y 133.038,Z 117.181,A -85,B 0,C 180,E1 -25417.957,E2 -25417.957} C_VEL
LIN {X 0,Y 134.198,Z 118.637,A -85,B 0,C 180,E1 -25418.82,E2 -25418.82} C_VEL
LIN {X 0,Y 137.969,Z 124.048,A -85,B 0,C 180,E1 -25421.47,E2 -25421.47} C_VEL
LIN {X 0,Y 142.864,Z 131.436,A -85,B 0,C 180,E1 -25424.529,E2 -25424.529} C_VEL
LIN {X 0,Y 148.763,Z 141.584,A -85,B 0,C 180,E1 -25427.822,E2 -25427.822} C_VEL
LIN {X 0,Y 154.114,Z 152.753,A -85,B 0,C 180,E1 -25430.572,E2 -25430.572} C_VEL
LIN {X 0,Y 153.495,Z 163.869,A -85,B 0,C 180,E1 -25431.054,E2 -25431.054} C_VEL
LIN {X 0,Y 151.066,Z 197.878,A -85,B 0,C 180,E1 -25432.467,E2 -25432.467} C_VEL
LIN {X 0,Y 149.25,Z 211.534,A -85,B 0,C 180,E1 -25433.524,E2 -25433.524} C_VEL
LIN {X 0,Y 147.005,Z 223.752,A -85,B 0,C 180,E1 -25434.993,E2 -25434.993} C_VEL
LIN {X 0,Y 143.829,Z 236.304,A -85,B 0,C 180,E1 -25437.071,E2 -25437.071} C_VEL
LIN {X 0,Y 140.335,Z 247.479,A -85,B 0,C 180,E1 -25439.533,E2 -25439.533} C_VEL
LIN {X 0,Y 136.617,Z 257.56,A -85,B 0,C 180,E1 -25442.421,E2 -25442.421} C_VEL
LIN {X 0,Y 132.82,Z 266.647,A -85,B 0,C 180,E1 -25445.791,E2 -25445.791} C_VEL
LIN {X 0,Y 128.906,Z 275.494,A -85,B 0,C 180,E1 -25450.078,E2 -25450.078} C_VEL
LIN {X 0,Y 125.663,Z 282.614,A -85,B 0,C 180,E1 -25454.595,E2 -25454.595} C_VEL
LIN {X 0,Y 123.441,Z 287.423,A -85,B 0,C 180,E1 -25458.507,E2 -25458.507} C_VEL
LIN {X 0,Y 121.459,Z 292.099,A -85,B 0,C 180,E1 -25463.355,E2 -25463.355} C_VEL
LIN {X 0,Y 120.294,Z 295.674,A -85,B 0,C 180,E1 -25468.327,E2 -25468.327} C_VEL
LIN {X 0,Y 119.734,Z 298.419,A -85,B 0,C 180,E1 -25473.744,E2 -25473.744} C_VEL
LIN {X 0,Y 119.578,Z 300.294,A -85,B 0,C 180,E1 -25480.157,E2 -25480.157} C_VEL
LIN {X 0,Y 120.659,Z 300.712,A -85,B 0,C 180,E1 -25486.933,E2 -25486.933} C_VEL
LIN {X 0,Y 121.811,Z 300.34,A -85,B 0,C 180,E1 -25490.255,E2 -25490.255} C_VEL
LIN {X 0,Y 123.999,Z 299.057,A -85,B 0,C 180,E1 -25494.925,E2 -25494.925} C_VEL
LIN {X 0,Y 128.24,Z 295.71,A -85,B 0,C 180,E1 -25501.376,E2 -25501.376} C_VEL
LIN {X 0,Y 132.207,Z 292.066,A -85,B 0,C 180,E1 -25505.786,E2 -25505.786} C_VEL
LIN {X 0,Y 136.894,Z 287.265,A -85,B 0,C 180,E1 -25509.938,E2 -25509.938} C_VEL
LIN {X 0,Y 142.228,Z 281.201,A -85,B 0,C 180,E1 -25513.773,E2 -25513.773} C_VEL
LIN {X 0,Y 148.145,Z 273.611,A -85,B 0,C 180,E1 -25517.336,E2 -25517.336} C_VEL
LIN {X 0,Y 153.624,Z 265.288,A -85,B 0,C 180,E1 -25520.318,E2 -25520.318} C_VEL
LIN {X 0,Y 159.457,Z 255.142,A -85,B 0,C 180,E1 -25523.022,E2 -25523.022} C_VEL
LIN {X 0,Y 164.843,Z 244.241,A -85,B 0,C 180,E1 -25525.158,E2 -25525.158} C_VEL
LIN {X 0,Y 169.409,Z 232.8,A -85,B 0,C 180,E1 -25526.828,E2 -25526.828} C_VEL
LIN {X 0,Y 172.985,Z 221.048,A -85,B 0,C 180,E1 -25528.164,E2 -25528.164} C_VEL
LIN {X 0,Y 176.006,Z 208.148,A -85,B 0,C 180,E1 -25529.155,E2 -25529.155} C_VEL
LIN {X 0,Y 177.971,Z 194.535,A -85,B 0,C 180,E1 -25529.824,E2 -25529.824} C_VEL
LIN {X 0,Y 179.491,Z 176.207,A -85,B 0,C 180,E1 -25530.439,E2 -25530.439} C_VEL
LIN {X 0,Y 175.127,Z 167.519,A -85,B 0,C 180,E1 -25533.402,E2 -25533.402} C_VEL
LIN {X 0,Y 171.199,Z 160.503,A -85,B 0,C 180,E1 -25536.395,E2 -25536.395} C_VEL
LIN {X 0,Y 167.574,Z 154.55,A -85,B 0,C 180,E1 -25539.559,E2 -25539.559} C_VEL
LIN {X 0,Y 165.314,Z 151.043,A -85,B 0,C 180,E1 -25541.807,E2 -25541.807} C_VEL
LIN {X 0,Y 162.938,Z 147.391,A -85,B 0,C 180,E1 -25544.52,E2 -25544.52} C_VEL
LIN {X 0,Y 160.464,Z 143.516,A -85,B 0,C 180,E1 -25547.952,E2 -25547.952} C_VEL
LIN {X 0,Y 158.232,Z 140.743,A -85,B 0,C 180,E1 -25551.86,E2 -25551.86} C_VEL
LIN {X 0,Y 157.459,Z 138.634,A -85,B 0,C 180,E1 -25553.914,E2 -25553.914} C_VEL
LIN {X 0,Y 155.801,Z 137.179,A -85,B 0,C 180,E1 -25559.999,E2 -25559.999} C_VEL
LIN {X 0,Y 155.783,Z 137.557,A -85,B 0,C 180,E1 -25566.605,E2 -25566.605} C_VEL
LIN {X 0,Y 157.394,Z 138.882,A -85,B 0,C 180,E1 -25572.435,E2 -25572.435} C_VEL
LIN {X 0,Y 159.144,Z 142.269,A -85,B 0,C 180,E1 -25576.392,E2 -25576.392} C_VEL
LIN {X 0,Y 160.719,Z 144.029,A -85,B 0,C 180,E1 -25578.886,E2 -25578.886} C_VEL
LIN {X 0,Y 163.68,Z 148.859,A -85,B 0,C 180,E1 -25582.84,E2 -25582.84} C_VEL
LIN {X 0,Y 166.519,Z 154.376,A -85,B 0,C 180,E1 -25586.01,E2 -25586.01} C_VEL
LIN {X 0,Y 169.873,Z 161.186,A -85,B 0,C 180,E1 -25589.202,E2 -25589.202} C_VEL
LIN {X 0,Y 174.294,Z 171.374,A -85,B 0,C 180,E1 -25592.86,E2 -25592.86} C_VEL
LIN {X 0,Y 178.179,Z 181.705,A -85,B 0,C 180,E1 -25595.735,E2 -25595.735} C_VEL
LIN {X 0,Y 178.892,Z 183.927,A -85,B 0,C 180,E1 -25596.25,E2 -25596.25} C_VEL
LIN {X 0,Y 176.607,Z 208.477,A -85,B 0,C 180,E1 -25597.074,E2 -25597.074} C_VEL
LIN {X 0,Y 174.29,Z 221.237,A -85,B 0,C 180,E1 -25597.768,E2 -25597.768} C_VEL
LIN {X 0,Y 170.839,Z 234.154,A -85,B 0,C 180,E1 -25598.825,E2 -25598.825} C_VEL
LIN {X 0,Y 166.612,Z 245.825,A -85,B 0,C 180,E1 -25600.132,E2 -25600.132} C_VEL
LIN {X 0,Y 161.555,Z 257.101,A -85,B 0,C 180,E1 -25601.842,E2 -25601.842} C_VEL
LIN {X 0,Y 156.159,Z 267.276,A -85,B 0,C 180,E1 -25603.937,E2 -25603.937} C_VEL
LIN {X 0,Y 150.537,Z 276.441,A -85,B 0,C 180,E1 -25606.478,E2 -25606.478} C_VEL
LIN {X 0,Y 144.127,Z 285.385,A -85,B 0,C 180,E1 -25609.75,E2 -25609.75} C_VEL
LIN {X 0,Y 138.367,Z 292.606,A -85,B 0,C 180,E1 -25613.357,E2 -25613.357} C_VEL
LIN {X 0,Y 134.147,Z 297.498,A -85,B 0,C 180,E1 -25616.625,E2 -25616.625} C_VEL
LIN {X 0,Y 129.716,Z 302.277,A -85,B 0,C 180,E1 -25620.815,E2 -25620.815} C_VEL
LIN {X 0,Y 125.927,Z 305.956,A -85,B 0,C 180,E1 -25625.254,E2 -25625.254} C_VEL
LIN {X 0,Y 122.905,Z 308.641,A -85,B 0,C 180,E1 -25629.933,E2 -25629.933} C_VEL
LIN {X 0,Y 120.432,Z 310.82,A -85,B 0,C 180,E1 -25636.5,E2 -25636.5} C_VEL
LIN {X 0,Y 119.407,Z 311.364,A -85,B 0,C 180,E1 -25643.239,E2 -25643.239} C_VEL
LIN {X 0,Y 119.506,Z 310.67,A -85,B 0,C 180,E1 -25648.695,E2 -25648.695} C_VEL
LIN {X 0,Y 119.497,Z 310.012,A -85,B 0,C 180,E1 -25651.107,E2 -25651.107} C_VEL
LIN {X 0,Y 119.444,Z 307.601,A -85,B 0,C 180,E1 -25656.757,E2 -25656.757} C_VEL
LIN {X 0,Y 120.006,Z 304.376,A -85,B 0,C 180,E1 -25661.827,E2 -25661.827} C_VEL
LIN {X 0,Y 121.235,Z 300.06,A -85,B 0,C 180,E1 -25666.848,E2 -25666.848} C_VEL
LIN {X 0,Y 123.958,Z 293.539,A -85,B 0,C 180,E1 -25672.5,E2 -25672.5} C_VEL
LIN {X 0,Y 124.362,Z 292.452,A -85,B 0,C 180,E1 -25673.283,E2 -25673.283} C_VEL
LIN {X 0,Y 125.023,Z 289.252,A -85,B 0,C 180,E1 -25675.55,E2 -25675.55} C_VEL
LIN {X 0,Y 124.815,Z 283.617,A -85,B 0,C 180,E1 -25679.303,E2 -25679.303} C_VEL
LIN {X 0,Y 125.02,Z 277.439,A -85,B 0,C 180,E1 -25682.853,E2 -25682.853} C_VEL
LIN {X 0,Y 126.266,Z 273.338,A -85,B 0,C 180,E1 -25684.711,E2 -25684.711} C_VEL
LIN {X 0,Y 130.278,Z 264.238,A -85,B 0,C 180,E1 -25687.852,E2 -25687.852} C_VEL
LIN {X 0,Y 134.532,Z 253.212,A -85,B 0,C 180,E1 -25690.767,E2 -25690.767} C_VEL
LIN {X 0,Y 138.088,Z 242.391,A -85,B 0,C 180,E1 -25692.899,E2 -25692.899} C_VEL
LIN {X 0,Y 141.645,Z 229.359,A -85,B 0,C 180,E1 -25694.743,E2 -25694.743} C_VEL
LIN {X 0,Y 144.025,Z 216.744,A -85,B 0,C 180,E1 -25696.033,E2 -25696.033} C_VEL
LIN {X 0,Y 145.591,Z 203.949,A -85,B 0,C 180,E1 -25696.857,E2 -25696.857} C_VEL
LIN {X 0,Y 148.047,Z 168.298,A -85,B 0,C 180,E1 -25698.349,E2 -25698.349} C_VEL
LIN {X 0,Y 147.523,Z 158.876,A -85,B 0,C 180,E1 -25699.19,E2 -25699.19} C_VEL
LIN {X 0,Y 144.239,Z 149.315,A -85,B 0,C 180,E1 -25701.224,E2 -25701.224} C_VEL
LIN {X 0,Y 139.97,Z 139.272,A -85,B 0,C 180,E1 -25703.956,E2 -25703.956} C_VEL
LIN {X 0,Y 136.313,Z 131.707,A -85,B 0,C 180,E1 -25706.485,E2 -25706.485} C_VEL
LIN {X 0,Y 130.616,Z 123.347,A -85,B 0,C 180,E1 -25710.733,E2 -25710.733} C_VEL
LIN {X 0,Y 127.985,Z 119.655,A -85,B 0,C 180,E1 -25712.992,E2 -25712.992} C_VEL
LIN {X 0,Y 124.823,Z 115.763,A -85,B 0,C 180,E1 -25715.998,E2 -25715.998} C_VEL
LIN {X 0,Y 123.97,Z 114.391,A -85,B 0,C 180,E1 -25716.931,E2 -25716.931} C_VEL
LIN {X 0,Y 121.241,Z 111.759,A -85,B 0,C 180,E1 -25719.979,E2 -25719.979} C_VEL
LIN {X 0,Y 119.935,Z 109.029,A -85,B 0,C 180,E1 -25721.863,E2 -25721.863} C_VEL
LIN {X 0,Y 117.266,Z 107.396,A -85,B 0,C 180,E1 -25725.688,E2 -25725.688} C_VEL
LIN {X 0,Y 115.633,Z 104.534,A -85,B 0,C 180,E1 -25729.027,E2 -25729.027} C_VEL
LIN {X 0,Y 115.366,Z 103.098,A -85,B 0,C 180,E1 -25730.025,E2 -25730.025} C_VEL
LIN {X 0,Y 115.99,Z 103.035,A -85,B 0,C 180,E1 -25740.001,E2 -25740.001} C_VEL
LIN {X 0,Y 115.359,Z 103.096,A -85,B 0,C 180,E1 -25746.999,E2 -25746.999} C_VEL
LIN {X 0,Y 115.207,Z 103.104,A -85,B 0,C 180,E1 -25752.57,E2 -25752.57} C_VEL
LIN {X 0,Y 115.055,Z 103.334,A -85,B 0,C 180,E1 -25757.211,E2 -25757.211} C_VEL
LIN {X 0,Y 115.624,Z 105.353,A -85,B 0,C 180,E1 -25758.84,E2 -25758.84} C_VEL
LIN {X 0,Y 117.602,Z 107.824,A -85,B 0,C 180,E1 -25762.575,E2 -25762.575} C_VEL
LIN {X 0,Y 119.922,Z 109.229,A -85,B 0,C 180,E1 -25765.842,E2 -25765.842} C_VEL
LIN {X 0,Y 121.375,Z 112.054,A -85,B 0,C 180,E1 -25767.897,E2 -25767.897} C_VEL
LIN {X 0,Y 123.895,Z 114.418,A -85,B 0,C 180,E1 -25770.7,E2 -25770.7} C_VEL
LIN {X 0,Y 124.763,Z 115.72,A -85,B 0,C 180,E1 -25771.641,E2 -25771.641} C_VEL
LIN {X 0,Y 127.015,Z 118.738,A -85,B 0,C 180,E1 -25773.859,E2 -25773.859} C_VEL
LIN {X 0,Y 128.102,Z 119.953,A -85,B 0,C 180,E1 -25774.826,E2 -25774.826} C_VEL
LIN {X 0,Y 130.691,Z 123.555,A -85,B 0,C 180,E1 -25777.034,E2 -25777.034} C_VEL
LIN {X 0,Y 134.768,Z 129.577,A -85,B 0,C 180,E1 -25780.149,E2 -25780.149} C_VEL
LIN {X 0,Y 140.079,Z 137.906,A -85,B 0,C 180,E1 -25783.689,E2 -25783.689} C_VEL
LIN {X 0,Y 145.433,Z 147.727,A -85,B 0,C 180,E1 -25786.875,E2 -25786.875} C_VEL
LIN {X 0,Y 148.888,Z 155.152,A -85,B 0,C 180,E1 -25788.792,E2 -25788.792} C_VEL
LIN {X 0,Y 145.86,Z 197.908,A -85,B 0,C 180,E1 -25790.615,E2 -25790.615} C_VEL
LIN {X 0,Y 143.91,Z 211.937,A -85,B 0,C 180,E1 -25791.714,E2 -25791.714} C_VEL
LIN {X 0,Y 141.537,Z 224.131,A -85,B 0,C 180,E1 -25793.205,E2 -25793.205} C_VEL
LIN {X 0,Y 138.445,Z 235.883,A -85,B 0,C 180,E1 -25795.175,E2 -25795.175} C_VEL
LIN {X 0,Y 134.755,Z 247.195,A -85,B 0,C 180,E1 -25797.686,E2 -25797.686} C_VEL
LIN {X 0,Y 130.842,Z 257.404,A -85,B 0,C 180,E1 -25800.651,E2 -25800.651} C_VEL
LIN {X 0,Y 126.421,Z 267.394,A -85,B 0,C 180,E1 -25804.48,E2 -25804.48} C_VEL
LIN {X 0,Y 122.297,Z 276.169,A -85,B 0,C 180,E1 -25808.952,E2 -25808.952} C_VEL
LIN {X 0,Y 118.861,Z 283.21,A -85,B 0,C 180,E1 -25813.69,E2 -25813.69} C_VEL
LIN {X 0,Y 115.714,Z 289.636,A -85,B 0,C 180,E1 -25819.503,E2 -25819.503} C_VEL
LIN {X 0,Y 113.939,Z 293.881,A -85,B 0,C 180,E1 -25824.692,E2 -25824.692} C_VEL
LIN {X 0,Y 112.904,Z 297.078,A -85,B 0,C 180,E1 -25830.001,E2 -25830.001} C_VEL
LIN {X 0,Y 112.637,Z 298.673,A -85,B 0,C 180,E1 -25833.578,E2 -25833.578} C_VEL
LIN {X 0,Y 112.444,Z 299.881,A -85,B 0,C 180,E1 -25837.182,E2 -25837.182} C_VEL
LIN {X 0,Y 113.006,Z 301.029,A -85,B 0,C 180,E1 -25844.406,E2 -25844.406} C_VEL
LIN {X 0,Y 115.085,Z 300.625,A -85,B 0,C 180,E1 -25851.495,E2 -25851.495} C_VEL
LIN {X 0,Y 117.282,Z 299.441,A -85,B 0,C 180,E1 -25855.99,E2 -25855.99} C_VEL
LIN {X 0,Y 120.865,Z 296.903,A -85,B 0,C 180,E1 -25861.557,E2 -25861.557} C_VEL
LIN {X 0,Y 124.908,Z 293.566,A -85,B 0,C 180,E1 -25866.214,E2 -25866.214} C_VEL
LIN {X 0,Y 129.992,Z 288.845,A -85,B 0,C 180,E1 -25870.806,E2 -25870.806} C_VEL
LIN {X 0,Y 136.128,Z 282.349,A -85,B 0,C 180,E1 -25875.227,E2 -25875.227} C_VEL
LIN {X 0,Y 142.298,Z 274.938,A -85,B 0,C 180,E1 -25878.868,E2 -25878.868} C_VEL
LIN {X 0,Y 148.467,Z 266.195,A -85,B 0,C 180,E1 -25882.123,E2 -25882.123} C_VEL
LIN {X 0,Y 154.051,Z 257.056,A -85,B 0,C 180,E1 -25884.636,E2 -25884.636} C_VEL
LIN {X 0,Y 158.97,Z 247.798,A -85,B 0,C 180,E1 -25886.561,E2 -25886.561} C_VEL
LIN {X 0,Y 164.029,Z 236.301,A -85,B 0,C 180,E1 -25888.384,E2 -25888.384} C_VEL
LIN {X 0,Y 167.969,Z 224.844,A -85,B 0,C 180,E1 -25889.783,E2 -25889.783} C_VEL
LIN {X 0,Y 171.377,Z 211.74,A -85,B 0,C 180,E1 -25890.886,E2 -25890.886} C_VEL
LIN {X 0,Y 173.719,Z 198.403,A -85,B 0,C 180,E1 -25891.616,E2 -25891.616} C_VEL
LIN {X 0,Y 175.458,Z 179.412,A -85,B 0,C 180,E1 -25892.279,E2 -25892.279} C_VEL
LIN {X 0,Y 171.08,Z 170.478,A -85,B 0,C 180,E1 -25895.578,E2 -25895.578} C_VEL
LIN {X 0,Y 167.147,Z 163.49,A -85,B 0,C 180,E1 -25898.963,E2 -25898.963} C_VEL
LIN {X 0,Y 163.935,Z 158.026,A -85,B 0,C 180,E1 -25902.214,E2 -25902.214} C_VEL
